LIN {X 0,Y 342.242,Z 667.887,A -85,B 0,C 180,E1 16805.675,E2 16805.675} C_VEL
LIN {X 0,Y 344.093,Z 652.07,A -85,B 0,C 180,E1 16803.884,E2 16803.884} C_VEL
LIN {X 0,Y 345.94,Z 635.37,A -85,B 0,C 180,E1 16802.363,E2 16802.363} C_VEL
LIN {X 0,Y 347.673,Z 617.854,A -85,B 0,C 180,E1 16801.111,E2 16801.111} C_VEL
LIN {X 0,Y 349.271,Z 599.201,A -85,B 0,C 180,E1 16800.115,E2 16800.115} C_VEL
LIN {X 0,Y 350.382,Z 580.027,A -85,B 0,C 180,E1 16799.421,E2 16799.421} C_VEL
LIN {X 0,Y 355.845,Z 417.127,A -85,B 0,C 180,E1 16795.462,E2 16795.462} C_VEL
LIN {X 0,Y 353.483,Z 389.228,A -85,B 0,C 180,E1 16794.516,E2 16794.516} C_VEL
LIN {X 0,Y 357.131,Z 365.009,A -85,B 0,C 180,E1 16791.622,E2 16791.622} C_VEL
LIN {X 0,Y 349.632,Z 342.182,A -85,B 0,C 180,E1 16787.791,E2 16787.791} C_VEL
LIN {X 0,Y 342.112,Z 320.607,A -85,B 0,C 180,E1 16783.792,E2 16783.792} C_VEL
LIN {X 0,Y 337.938,Z 308.703,A -85,B 0,C 180,E1 16781.36,E2 16781.36} C_VEL
LIN {X 0,Y 337.929,Z 308.702,A -85,B 0,C 180,E1 16777.13,E2 16777.13} C_VEL
LIN {X 0,Y 337.924,Z 308.701,A -85,B 0,C 180,E1 16772.83,E2 16772.83} C_VEL
LIN {X 0,Y 337.928,Z 308.701,A -85,B 0,C 180,E1 16768.45,E2 16768.45} C_VEL
LIN {X 0,Y 337.933,Z 308.701,A -85,B 0,C 180,E1 16764.286,E2 16764.286} C_VEL
LIN {X 0,Y 337.943,Z 308.701,A -85,B 0,C 180,E1 16760.074,E2 16760.074} C_VEL
LIN {X 0,Y 337.961,Z 308.701,A -85,B 0,C 180,E1 16755.796,E2 16755.796} C_VEL
LIN {X 0,Y 337.96,Z 308.702,A -85,B 0,C 180,E1 16751.608,E2 16751.608} C_VEL
LIN {X 0,Y 337.954,Z 308.7,A -85,B 0,C 180,E1 16747.311,E2 16747.311} C_VEL
LIN {X 0,Y 337.939,Z 308.699,A -85,B 0,C 180,E1 16743.055,E2 16743.055} C_VEL
LIN {X 0,Y 337.933,Z 308.7,A -85,B 0,C 180,E1 16738.816,E2 16738.816} C_VEL
LIN {X 0,Y 337.931,Z 308.7,A -85,B 0,C 180,E1 16734.57,E2 16734.57} C_VEL
LIN {X 0,Y 337.934,Z 308.699,A -85,B 0,C 180,E1 16730.293,E2 16730.293} C_VEL
LIN {X 0,Y 337.947,Z 308.7,A -85,B 0,C 180,E1 16726.025,E2 16726.025} C_VEL
LIN {X 0,Y 337.963,Z 308.7,A -85,B 0,C 180,E1 16721.727,E2 16721.727} C_VEL
LIN {X 0,Y 337.977,Z 308.698,A -85,B 0,C 180,E1 16717.366,E2 16717.366} C_VEL
LIN {X 0,Y 337.959,Z 308.697,A -85,B 0,C 180,E1 16713.089,E2 16713.089} C_VEL
LIN {X 0,Y 337.958,Z 308.697,A -85,B 0,C 180,E1 16709.021,E2 16709.021} C_VEL
LIN {X 0,Y 337.945,Z 308.698,A -85,B 0,C 180,E1 16704.742,E2 16704.742} C_VEL
LIN {X 0,Y 337.941,Z 308.697,A -85,B 0,C 180,E1 16700.501,E2 16700.501} C_VEL
LIN {X 0,Y 337.944,Z 308.698,A -85,B 0,C 180,E1 16696.19,E2 16696.19} C_VEL
LIN {X 0,Y 337.951,Z 308.699,A -85,B 0,C 180,E1 16691.96,E2 16691.96} C_VEL
LIN {X 0,Y 337.96,Z 308.698,A -85,B 0,C 180,E1 16687.762,E2 16687.762} C_VEL
LIN {X 0,Y 337.98,Z 308.699,A -85,B 0,C 180,E1 16683.382,E2 16683.382} C_VEL
LIN {X 0,Y 337.989,Z 308.696,A -85,B 0,C 180,E1 16679.215,E2 16679.215} C_VEL
LIN {X 0,Y 337.962,Z 308.695,A -85,B 0,C 180,E1 16674.84,E2 16674.84} C_VEL
LIN {X 0,Y 337.954,Z 308.697,A -85,B 0,C 180,E1 16670.612,E2 16670.612} C_VEL
LIN {X 0,Y 337.948,Z 308.697,A -85,B 0,C 180,E1 16666.323,E2 16666.323} C_VEL
LIN {X 0,Y 337.95,Z 308.697,A -85,B 0,C 180,E1 16662.125,E2 16662.125} C_VEL
LIN {X 0,Y 337.957,Z 308.699,A -85,B 0,C 180,E1 16657.82,E2 16657.82} C_VEL
LIN {X 0,Y 337.97,Z 308.699,A -85,B 0,C 180,E1 16653.561,E2 16653.561} C_VEL
LIN {X 0,Y 337.989,Z 308.698,A -85,B 0,C 180,E1 16649.321,E2 16649.321} C_VEL
LIN {X 0,Y 337.976,Z 308.696,A -85,B 0,C 180,E1 16644.907,E2 16644.907} C_VEL
LIN {X 0,Y 337.973,Z 308.695,A -85,B 0,C 180,E1 16640.806,E2 16640.806} C_VEL
LIN {X 0,Y 337.96,Z 308.696,A -85,B 0,C 180,E1 16636.482,E2 16636.482} C_VEL
LIN {X 0,Y 337.959,Z 308.696,A -85,B 0,C 180,E1 16632.257,E2 16632.257} C_VEL
LIN {X 0,Y 337.957,Z 308.698,A -85,B 0,C 180,E1 16627.929,E2 16627.929} C_VEL
LIN {X 0,Y 337.97,Z 308.698,A -85,B 0,C 180,E1 16623.654,E2 16623.654} C_VEL
LIN {X 0,Y 337.982,Z 308.699,A -85,B 0,C 180,E1 16619.407,E2 16619.407} C_VEL
LIN {X 0,Y 337.987,Z 308.698,A -85,B 0,C 180,E1 16615.182,E2 16615.182} C_VEL
LIN {X 0,Y 337.991,Z 308.694,A -85,B 0,C 180,E1 16610.805,E2 16610.805} C_VEL
LIN {X 0,Y 337.978,Z 308.696,A -85,B 0,C 180,E1 16606.658,E2 16606.658} C_VEL
LIN {X 0,Y 337.971,Z 308.699,A -85,B 0,C 180,E1 16602.412,E2 16602.412} C_VEL
LIN {X 0,Y 337.978,Z 308.752,A -85,B 0,C 180,E1 16601.593,E2 16601.593} C_VEL
LIN {X 0,Y 342.926,Z 325.779,A -85,B 0,C 180,E1 16597.751,E2 16597.751} C_VEL
LIN {X 0,Y 347.577,Z 343.263,A -85,B 0,C 180,E1 16594.056,E2 16594.056} C_VEL
LIN {X 0,Y 349.757,Z 352.134,A -85,B 0,C 180,E1 16592.257,E2 16592.257} C_VEL
LIN {X 0,Y 349.677,Z 355.829,A -85,B 0,C 180,E1 16591.603,E2 16591.603} C_VEL
LIN {X 0,Y 347.871,Z 360.579,A -85,B 0,C 180,E1 16590.902,E2 16590.902} C_VEL
LIN {X 0,Y 340.468,Z 373.577,A -85,B 0,C 180,E1 16589.15,E2 16589.15} C_VEL
LIN {X 0,Y 339.309,Z 377.653,A -85,B 0,C 180,E1 16588.506,E2 16588.506} C_VEL
LIN {X 0,Y 336.591,Z 401.793,A -85,B 0,C 180,E1 16584.466,E2 16584.466} C_VEL
LIN {X 0,Y 340.456,Z 436.456,A -85,B 0,C 180,E1 16583.068,E2 16583.068} C_VEL
LIN {X 0,Y 336.471,Z 532.966,A -85,B 0,C 180,E1 16580.059,E2 16580.059} C_VEL
LIN {X 0,Y 335.72,Z 549.826,A -85,B 0,C 180,E1 16579.22,E2 16579.22} C_VEL
LIN {X 0,Y 334.81,Z 566.067,A -85,B 0,C 180,E1 16578.091,E2 16578.091} C_VEL
LIN {X 0,Y 333.738,Z 582.038,A -85,B 0,C 180,E1 16576.622,E2 16576.622} C_VEL
LIN {X 0,Y 332.698,Z 596.678,A -85,B 0,C 180,E1 16574.886,E2 16574.886} C_VEL
LIN {X 0,Y 331.716,Z 609.954,A -85,B 0,C 180,E1 16572.885,E2 16572.885} C_VEL
LIN {X 0,Y 330.934,Z 620.947,A -85,B 0,C 180,E1 16570.794,E2 16570.794} C_VEL
LIN {X 0,Y 330.399,Z 629.807,A -85,B 0,C 180,E1 16568.7,E2 16568.7} C_VEL
LIN {X 0,Y 330.037,Z 637.83,A -85,B 0,C 180,E1 16566.259,E2 16566.259} C_VEL
LIN {X 0,Y 329.915,Z 643.784,A -85,B 0,C 180,E1 16563.82,E2 16563.82} C_VEL
LIN {X 0,Y 330.037,Z 648.132,A -85,B 0,C 180,E1 16561.241,E2 16561.241} C_VEL
LIN {X 0,Y 330.399,Z 650.527,A -85,B 0,C 180,E1 16558.61,E2 16558.61} C_VEL
LIN {X 0,Y 330.992,Z 651.065,A -85,B 0,C 180,E1 16556.187,E2 16556.187} C_VEL
LIN {X 0,Y 331.918,Z 649.726,A -85,B 0,C 180,E1 16553.598,E2 16553.598} C_VEL
LIN {X 0,Y 333.117,Z 646.807,A -85,B 0,C 180,E1 16551.192,E2 16551.192} C_VEL
LIN {X 0,Y 334.647,Z 642.03,A -85,B 0,C 180,E1 16548.799,E2 16548.799} C_VEL
LIN {X 0,Y 336.587,Z 635.419,A -85,B 0,C 180,E1 16546.425,E2 16546.425} C_VEL
LIN {X 0,Y 338.907,Z 626.513,A -85,B 0,C 180,E1 16544.073,E2 16544.073} C_VEL
LIN {X 0,Y 341.25,Z 616.897,A -85,B 0,C 180,E1 16542.08,E2 16542.08} C_VEL
LIN {X 0,Y 343.89,Z 604.887,A -85,B 0,C 180,E1 16540.11,E2 16540.11} C_VEL
LIN {X 0,Y 346.665,Z 591.244,A -85,B 0,C 180,E1 16538.333,E2 16538.333} C_VEL
LIN {X 0,Y 349.446,Z 575.669,A -85,B 0,C 180,E1 16536.741,E2 16536.741} C_VEL
LIN {X 0,Y 351.92,Z 559.982,A -85,B 0,C 180,E1 16535.491,E2 16535.491} C_VEL
LIN {X 0,Y 354.216,Z 542.534,A -85,B 0,C 180,E1 16534.445,E2 16534.445} C_VEL
LIN {X 0,Y 361.198,Z 491.904,A -85,B 0,C 180,E1 16532.223,E2 16532.223} C_VEL
LIN {X 0,Y 367.897,Z 448.392,A -85,B 0,C 180,E1 16530.39,E2 16530.39} C_VEL
LIN {X 0,Y 367.465,Z 432.669,A -85,B 0,C 180,E1 16528.882,E2 16528.882} C_VEL
LIN {X 0,Y 366.778,Z 418.433,A -85,B 0,C 180,E1 16527.238,E2 16527.238} C_VEL
LIN {X 0,Y 366.27,Z 405.199,A -85,B 0,C 180,E1 16525.43,E2 16525.43} C_VEL
LIN {X 0,Y 366.35,Z 400.175,A -85,B 0,C 180,E1 16524.646,E2 16524.646} C_VEL
LIN {X 0,Y 368.778,Z 395.594,A -85,B 0,C 180,E1 16523.573,E2 16523.573} C_VEL
LIN {X 0,Y 369.415,Z 391.695,A -85,B 0,C 180,E1 16521.299,E2 16521.299} C_VEL
LIN {X 0,Y 370.024,Z 389.528,A -85,B 0,C 180,E1 16518.931,E2 16518.931} C_VEL
LIN {X 0,Y 370.832,Z 389.284,A -85,B 0,C 180,E1 16516.495,E2 16516.495} C_VEL
LIN {X 0,Y 371.534,Z 391.679,A -85,B 0,C 180,E1 16513.974,E2 16513.974} C_VEL
LIN {X 0,Y 372.084,Z 395.125,A -85,B 0,C 180,E1 16512.103,E2 16512.103} C_VEL
LIN {X 0,Y 371.235,Z 397.302,A -85,B 0,C 180,E1 16511.78,E2 16511.78} C_VEL
LIN {X 0,Y 371.46,Z 412.671,A -85,B 0,C 180,E1 16510.389,E2 16510.389} C_VEL
LIN {X 0,Y 371.239,Z 424.916,A -85,B 0,C 180,E1 16509.557,E2 16509.557} C_VEL
LIN {X 0,Y 362.025,Z 501.522,A -85,B 0,C 180,E1 16507.037,E2 16507.037} C_VEL
LIN {X 0,Y 354.62,Z 580.346,A -85,B 0,C 180,E1 16504.536,E2 16504.536} C_VEL
LIN {X 0,Y 351.887,Z 599.701,A -85,B 0,C 180,E1 16503.638,E2 16503.638} C_VEL
LIN {X 0,Y 348.616,Z 618.561,A -85,B 0,C 180,E1 16502.436,E2 16502.436} C_VEL
LIN {X 0,Y 345.167,Z 636.473,A -85,B 0,C 180,E1 16500.943,E2 16500.943} C_VEL
LIN {X 0,Y 341.679,Z 653.443,A -85,B 0,C 180,E1 16499.15,E2 16499.15} C_VEL
LIN {X 0,Y 338.323,Z 669.249,A -85,B 0,C 180,E1 16497.074,E2 16497.074} C_VEL
LIN {X 0,Y 335.124,Z 684.622,A -85,B 0,C 180,E1 16494.597,E2 16494.597} C_VEL
LIN {X 0,Y 332.517,Z 698.311,A -85,B 0,C 180,E1 16491.893,E2 16491.893} C_VEL
LIN {X 0,Y 330.578,Z 709.97,A -85,B 0,C 180,E1 16489.067,E2 16489.067} C_VEL
LIN {X 0,Y 329.306,Z 720.112,A -85,B 0,C 180,E1 16486.041,E2 16486.041} C_VEL
LIN {X 0,Y 328.706,Z 728.665,A -85,B 0,C 180,E1 16482.831,E2 16482.831} C_VEL
LIN {X 0,Y 328.709,Z 735.179,A -85,B 0,C 180,E1 16479.632,E2 16479.632} C_VEL
LIN {X 0,Y 329.047,Z 739.533,A -85,B 0,C 180,E1 16476.632,E2 16476.632} C_VEL
LIN {X 0,Y 329.486,Z 742.179,A -85,B 0,C 180,E1 16473.655,E2 16473.655} C_VEL
LIN {X 0,Y 329.775,Z 743.096,A -85,B 0,C 180,E1 16470.87,E2 16470.87} C_VEL
LIN {X 0,Y 329.767,Z 742.439,A -85,B 0,C 180,E1 16468.09,E2 16468.09} C_VEL
LIN {X 0,Y 329.514,Z 740.182,A -85,B 0,C 180,E1 16465.302,E2 16465.302} C_VEL
LIN {X 0,Y 329.182,Z 736.275,A -85,B 0,C 180,E1 16462.497,E2 16462.497} C_VEL
LIN {X 0,Y 328.954,Z 730.625,A -85,B 0,C 180,E1 16459.671,E2 16459.671} C_VEL
LIN {X 0,Y 329.017,Z 723.102,A -85,B 0,C 180,E1 16456.827,E2 16456.827} C_VEL
LIN {X 0,Y 329.447,Z 714.162,A -85,B 0,C 180,E1 16454.15,E2 16454.15} C_VEL
LIN {X 0,Y 330.336,Z 703.098,A -85,B 0,C 180,E1 16451.471,E2 16451.471} C_VEL
LIN {X 0,Y 331.632,Z 690.48,A -85,B 0,C 180,E1 16448.976,E2 16448.976} C_VEL
LIN {X 0,Y 333.279,Z 676.261,A -85,B 0,C 180,E1 16446.673,E2 16446.673} C_VEL
LIN {X 0,Y 335.14,Z 660.941,A -85,B 0,C 180,E1 16444.653,E2 16444.653} C_VEL
LIN {X 0,Y 337.069,Z 644.579,A -85,B 0,C 180,E1 16442.915,E2 16442.915} C_VEL
LIN {X 0,Y 338.953,Z 627.296,A -85,B 0,C 180,E1 16441.455,E2 16441.455} C_VEL
LIN {X 0,Y 340.72,Z 609.034,A -85,B 0,C 180,E1 16440.27,E2 16440.27} C_VEL
LIN {X 0,Y 342.192,Z 590.096,A -85,B 0,C 180,E1 16439.383,E2 16439.383} C_VEL
LIN {X 0,Y 343.081,Z 569.712,A -85,B 0,C 180,E1 16438.771,E2 16438.771} C_VEL
LIN {X 0,Y 348.452,Z 418.182,A -85,B 0,C 180,E1 16434.993,E2 16434.993} C_VEL
LIN {X 0,Y 346.093,Z 389.328,A -85,B 0,C 180,E1 16433.992,E2 16433.992} C_VEL
LIN {X 0,Y 349.501,Z 367.033,A -85,B 0,C 180,E1 16431.259,E2 16431.259} C_VEL
LIN {X 0,Y 342.384,Z 345.277,A -85,B 0,C 180,E1 16427.523,E2 16427.523} C_VEL
LIN {X 0,Y 335.056,Z 324.104,A -85,B 0,C 180,E1 16423.521,E2 16423.521} C_VEL
LIN {X 0,Y 329.981,Z 309.695,A -85,B 0,C 180,E1 16420.539,E2 16420.539} C_VEL
LIN {X 0,Y 329.992,Z 309.692,A -85,B 0,C 180,E1 16416.219,E2 16416.219} C_VEL
LIN {X 0,Y 330.019,Z 309.691,A -85,B 0,C 180,E1 16411.816,E2 16411.816} C_VEL
LIN {X 0,Y 330.02,Z 309.69,A -85,B 0,C 180,E1 16407.618,E2 16407.618} C_VEL
LIN {X 0,Y 330.01,Z 309.69,A -85,B 0,C 180,E1 16403.365,E2 16403.365} C_VEL
LIN {X 0,Y 329.999,Z 309.69,A -85,B 0,C 180,E1 16399.103,E2 16399.103} C_VEL
LIN {X 0,Y 329.986,Z 309.69,A -85,B 0,C 180,E1 16394.747,E2 16394.747} C_VEL
LIN {X 0,Y 329.995,Z 309.69,A -85,B 0,C 180,E1 16390.3,E2 16390.3} C_VEL
LIN {X 0,Y 330.003,Z 309.69,A -85,B 0,C 180,E1 16386.09,E2 16386.09} C_VEL
LIN {X 0,Y 330.022,Z 309.69,A -85,B 0,C 180,E1 16381.739,E2 16381.739} C_VEL
LIN {X 0,Y 330.02,Z 309.688,A -85,B 0,C 180,E1 16377.398,E2 16377.398} C_VEL
LIN {X 0,Y 330.005,Z 309.688,A -85,B 0,C 180,E1 16373.042,E2 16373.042} C_VEL
LIN {X 0,Y 329.998,Z 309.687,A -85,B 0,C 180,E1 16368.822,E2 16368.822} C_VEL
LIN {X 0,Y 329.996,Z 309.689,A -85,B 0,C 180,E1 16364.469,E2 16364.469} C_VEL
LIN {X 0,Y 330.003,Z 309.686,A -85,B 0,C 180,E1 16360.166,E2 16360.166} C_VEL
LIN {X 0,Y 330.008,Z 309.689,A -85,B 0,C 180,E1 16356.05,E2 16356.05} C_VEL
LIN {X 0,Y 330.022,Z 309.687,A -85,B 0,C 180,E1 16351.798,E2 16351.798} C_VEL
LIN {X 0,Y 330.034,Z 309.688,A -85,B 0,C 180,E1 16347.576,E2 16347.576} C_VEL
LIN {X 0,Y 330.025,Z 309.686,A -85,B 0,C 180,E1 16343.144,E2 16343.144} C_VEL
LIN {X 0,Y 330.015,Z 309.683,A -85,B 0,C 180,E1 16338.899,E2 16338.899} C_VEL
LIN {X 0,Y 330.007,Z 309.687,A -85,B 0,C 180,E1 16334.607,E2 16334.607} C_VEL
LIN {X 0,Y 330.006,Z 309.687,A -85,B 0,C 180,E1 16330.19,E2 16330.19} C_VEL
LIN {X 0,Y 330.011,Z 309.684,A -85,B 0,C 180,E1 16325.998,E2 16325.998} C_VEL
LIN {X 0,Y 330.031,Z 309.688,A -85,B 0,C 180,E1 16321.652,E2 16321.652} C_VEL
LIN {X 0,Y 330.044,Z 309.686,A -85,B 0,C 180,E1 16317.416,E2 16317.416} C_VEL
LIN {X 0,Y 330.034,Z 309.684,A -85,B 0,C 180,E1 16313.004,E2 16313.004} C_VEL
LIN {X 0,Y 330.02,Z 309.686,A -85,B 0,C 180,E1 16308.731,E2 16308.731} C_VEL
LIN {X 0,Y 330.009,Z 309.685,A -85,B 0,C 180,E1 16304.384,E2 16304.384} C_VEL
LIN {X 0,Y 330.015,Z 309.687,A -85,B 0,C 180,E1 16299.943,E2 16299.943} C_VEL
LIN {X 0,Y 330.023,Z 309.688,A -85,B 0,C 180,E1 16295.737,E2 16295.737} C_VEL
LIN {X 0,Y 330.041,Z 309.688,A -85,B 0,C 180,E1 16291.387,E2 16291.387} C_VEL
LIN {X 0,Y 330.04,Z 309.684,A -85,B 0,C 180,E1 16287.047,E2 16287.047} C_VEL
LIN {X 0,Y 330.029,Z 309.685,A -85,B 0,C 180,E1 16282.688,E2 16282.688} C_VEL
LIN {X 0,Y 330.019,Z 309.685,A -85,B 0,C 180,E1 16278.464,E2 16278.464} C_VEL
LIN {X 0,Y 330.017,Z 309.685,A -85,B 0,C 180,E1 16274.175,E2 16274.175} C_VEL
LIN {X 0,Y 330.024,Z 309.687,A -85,B 0,C 180,E1 16269.794,E2 16269.794} C_VEL
LIN {X 0,Y 330.029,Z 309.688,A -85,B 0,C 180,E1 16265.666,E2 16265.666} C_VEL
LIN {X 0,Y 330.045,Z 309.688,A -85,B 0,C 180,E1 16261.401,E2 16261.401} C_VEL
LIN {X 0,Y 330.053,Z 309.685,A -85,B 0,C 180,E1 16257.043,E2 16257.043} C_VEL
LIN {X 0,Y 330.042,Z 309.684,A -85,B 0,C 180,E1 16252.705,E2 16252.705} C_VEL
LIN {X 0,Y 330.032,Z 309.685,A -85,B 0,C 180,E1 16248.433,E2 16248.433} C_VEL
LIN {X 0,Y 330.026,Z 309.69,A -85,B 0,C 180,E1 16244.107,E2 16244.107} C_VEL
LIN {X 0,Y 330.047,Z 309.82,A -85,B 0,C 180,E1 16242.293,E2 16242.293} C_VEL
LIN {X 0,Y 335.328,Z 327.903,A -85,B 0,C 180,E1 16238.109,E2 16238.109} C_VEL
LIN {X 0,Y 340.028,Z 345.65,A -85,B 0,C 180,E1 16234.279,E2 16234.279} C_VEL
LIN {X 0,Y 342.178,Z 355.277,A -85,B 0,C 180,E1 16232.322,E2 16232.322} C_VEL
LIN {X 0,Y 339.309,Z 377.653,A -85,B 0,C 180,E1 16228.506,E2 16228.506} C_VEL
LIN {X 0,Y 337.908,Z 381.407,A -85,B 0,C 180,E1 16227.937,E2 16227.937} C_VEL
LIN {X 0,Y 330.822,Z 391.443,A -85,B 0,C 180,E1 16226.626,E2 16226.626} C_VEL
LIN {X 0,Y 329.73,Z 394.679,A -85,B 0,C 180,E1 16226.118,E2 16226.118} C_VEL
LIN {X 0,Y 328.981,Z 401.707,A -85,B 0,C 180,E1 16224.957,E2 16224.957} C_VEL
LIN {X 0,Y 332.841,Z 437.209,A -85,B 0,C 180,E1 16223.481,E2 16223.481} C_VEL
LIN {X 0,Y 328.703,Z 533.627,A -85,B 0,C 180,E1 16220.38,E2 16220.38} C_VEL
LIN {X 0,Y 327.948,Z 550.028,A -85,B 0,C 180,E1 16219.546,E2 16219.546} C_VEL
LIN {X 0,Y 326.976,Z 566.748,A -85,B 0,C 180,E1 16218.356,E2 16218.356} C_VEL
LIN {X 0,Y 325.863,Z 582.787,A -85,B 0,C 180,E1 16216.843,E2 16216.843} C_VEL
LIN {X 0,Y 324.745,Z 598.018,A -85,B 0,C 180,E1 16214.986,E2 16214.986} C_VEL
LIN {X 0,Y 323.745,Z 611.255,A -85,B 0,C 180,E1 16212.936,E2 16212.936} C_VEL
LIN {X 0,Y 322.93,Z 622.663,A -85,B 0,C 180,E1 16210.703,E2 16210.703} C_VEL
LIN {X 0,Y 322.402,Z 631.415,A -85,B 0,C 180,E1 16208.558,E2 16208.558} C_VEL
LIN {X 0,Y 322.064,Z 639.424,A -85,B 0,C 180,E1 16206.056,E2 16206.056} C_VEL
LIN {X 0,Y 321.969,Z 645.288,A -85,B 0,C 180,E1 16203.558,E2 16203.558} C_VEL
LIN {X 0,Y 322.12,Z 649.393,A -85,B 0,C 180,E1 16201.065,E2 16201.065} C_VEL
LIN {X 0,Y 322.531,Z 651.846,A -85,B 0,C 180,E1 16198.399,E2 16198.399} C_VEL
LIN {X 0,Y 323.192,Z 652.469,A -85,B 0,C 180,E1 16195.917,E2 16195.917} C_VEL
LIN {X 0,Y 324.223,Z 651.242,A -85,B 0,C 180,E1 16193.268,E2 16193.268} C_VEL
LIN {X 0,Y 325.534,Z 648.402,A -85,B 0,C 180,E1 16190.807,E2 16190.807} C_VEL
LIN {X 0,Y 327.224,Z 643.805,A -85,B 0,C 180,E1 16188.363,E2 16188.363} C_VEL
LIN {X 0,Y 329.322,Z 637.306,A -85,B 0,C 180,E1 16185.941,E2 16185.941} C_VEL
LIN {X 0,Y 331.657,Z 629.375,A -85,B 0,C 180,E1 16183.716,E2 16183.716} C_VEL
LIN {X 0,Y 334.367,Z 619.283,A -85,B 0,C 180,E1 16181.518,E2 16181.518} C_VEL
LIN {X 0,Y 337.349,Z 607.161,A -85,B 0,C 180,E1 16179.436,E2 16179.436} C_VEL
LIN {X 0,Y 340.615,Z 592.522,A -85,B 0,C 180,E1 16177.474,E2 16177.474} C_VEL
LIN {X 0,Y 343.465,Z 578.024,A -85,B 0,C 180,E1 16175.947,E2 16175.947} C_VEL
LIN {X 0,Y 346.281,Z 561.82,A -85,B 0,C 180,E1 16174.608,E2 16174.608} C_VEL
LIN {X 0,Y 348.857,Z 544.428,A -85,B 0,C 180,E1 16173.52,E2 16173.52} C_VEL
LIN {X 0,Y 355.467,Z 499.569,A -85,B 0,C 180,E1 16171.483,E2 16171.483} C_VEL
LIN {X 0,Y 363.522,Z 450.722,A -85,B 0,C 180,E1 16169.389,E2 16169.389} C_VEL
LIN {X 0,Y 363.468,Z 436.002,A -85,B 0,C 180,E1 16167.918,E2 16167.918} C_VEL
LIN {X 0,Y 363.231,Z 422.494,A -85,B 0,C 180,E1 16166.301,E2 16166.301} C_VEL
LIN {X 0,Y 363.194,Z 409.998,A -85,B 0,C 180,E1 16164.539,E2 16164.539} C_VEL
LIN {X 0,Y 363.472,Z 400.515,A -85,B 0,C 180,E1 16162.954,E2 16162.954} C_VEL
LIN {X 0,Y 363.94,Z 397.554,A -85,B 0,C 180,E1 16161.214,E2 16161.214} C_VEL
LIN {X 0,Y 364.674,Z 395.498,A -85,B 0,C 180,E1 16158.939,E2 16158.939} C_VEL
LIN {X 0,Y 365.497,Z 395.214,A -85,B 0,C 180,E1 16156.633,E2 16156.633} C_VEL
LIN {X 0,Y 366.141,Z 397.534,A -85,B 0,C 180,E1 16154.111,E2 16154.111} C_VEL
LIN {X 0,Y 367.925,Z 401.188,A -85,B 0,C 180,E1 16152.735,E2 16152.735} C_VEL
LIN {X 0,Y 367.706,Z 416.125,A -85,B 0,C 180,E1 16151.346,E2 16151.346} C_VEL
LIN {X 0,Y 367.217,Z 426.833,A -85,B 0,C 180,E1 16150.599,E2 16150.599} C_VEL
LIN {X 0,Y 357.366,Z 500.917,A -85,B 0,C 180,E1 16148.093,E2 16148.093} C_VEL
LIN {X 0,Y 349.11,Z 579.334,A -85,B 0,C 180,E1 16145.506,E2 16145.506} C_VEL
LIN {X 0,Y 346.376,Z 597.432,A -85,B 0,C 180,E1 16144.659,E2 16144.659} C_VEL
LIN {X 0,Y 342.837,Z 616.357,A -85,B 0,C 180,E1 16143.451,E2 16143.451} C_VEL
LIN {X 0,Y 339.114,Z 634.228,A -85,B 0,C 180,E1 16141.956,E2 16141.956} C_VEL
LIN {X 0,Y 335.36,Z 651.175,A -85,B 0,C 180,E1 16140.158,E2 16140.158} C_VEL
LIN {X 0,Y 331.681,Z 667.065,A -85,B 0,C 180,E1 16138.053,E2 16138.053} C_VEL
LIN {X 0,Y 328.265,Z 681.983,A -85,B 0,C 180,E1 16135.629,E2 16135.629} C_VEL
LIN {X 0,Y 325.403,Z 695.384,A -85,B 0,C 180,E1 16132.97,E2 16132.97} C_VEL
LIN {X 0,Y 323.16,Z 707.314,A -85,B 0,C 180,E1 16130.088,E2 16130.088} C_VEL
LIN {X 0,Y 321.607,Z 717.69,A -85,B 0,C 180,E1 16126.993,E2 16126.993} C_VEL
LIN {X 0,Y 320.831,Z 726.031,A -85,B 0,C 180,E1 16123.886,E2 16123.886} C_VEL
LIN {X 0,Y 320.66,Z 732.543,A -85,B 0,C 180,E1 16120.784,E2 16120.784} C_VEL
LIN {X 0,Y 320.939,Z 737.326,A -85,B 0,C 180,E1 16117.7,E2 16117.7} C_VEL
LIN {X 0,Y 321.411,Z 740.407,A -85,B 0,C 180,E1 16114.641,E2 16114.641} C_VEL
LIN {X 0,Y 321.79,Z 741.759,A -85,B 0,C 180,E1 16111.782,E2 16111.782} C_VEL
LIN {X 0,Y 321.918,Z 741.55,A -85,B 0,C 180,E1 16109.112,E2 16109.112} C_VEL
LIN {X 0,Y 321.729,Z 739.777,A -85,B 0,C 180,E1 16106.259,E2 16106.259} C_VEL
LIN {X 0,Y 321.381,Z 736.362,A -85,B 0,C 180,E1 16103.391,E2 16103.391} C_VEL
LIN {X 0,Y 321.083,Z 731.227,A -85,B 0,C 180,E1 16100.502,E2 16100.502} C_VEL
LIN {X 0,Y 321.024,Z 724.256,A -85,B 0,C 180,E1 16097.591,E2 16097.591} C_VEL
LIN {X 0,Y 321.36,Z 715.365,A -85,B 0,C 180,E1 16094.695,E2 16094.695} C_VEL
LIN {X 0,Y 322.159,Z 704.733,A -85,B 0,C 180,E1 16091.92,E2 16091.92} C_VEL
LIN {X 0,Y 323.384,Z 692.644,A -85,B 0,C 180,E1 16089.363,E2 16089.363} C_VEL
LIN {X 0,Y 324.962,Z 679.01,A -85,B 0,C 180,E1 16087,E2 16087} C_VEL
LIN {X 0,Y 326.848,Z 663.752,A -85,B 0,C 180,E1 16084.837,E2 16084.837} C_VEL
LIN {X 0,Y 328.807,Z 647.754,A -85,B 0,C 180,E1 16082.999,E2 16082.999} C_VEL
LIN {X 0,Y 330.729,Z 631.142,A -85,B 0,C 180,E1 16081.469,E2 16081.469} C_VEL
LIN {X 0,Y 332.604,Z 612.794,A -85,B 0,C 180,E1 16080.166,E2 16080.166} C_VEL
LIN {X 0,Y 334.19,Z 594.034,A -85,B 0,C 180,E1 16079.191,E2 16079.191} C_VEL
LIN {X 0,Y 335.235,Z 574.913,A -85,B 0,C 180,E1 16078.52,E2 16078.52} C_VEL
LIN {X 0,Y 340.999,Z 418.598,A -85,B 0,C 180,E1 16074.49,E2 16074.49} C_VEL
LIN {X 0,Y 338.72,Z 389.414,A -85,B 0,C 180,E1 16073.451,E2 16073.451} C_VEL
LIN {X 0,Y 341.939,Z 369.272,A -85,B 0,C 180,E1 16070.929,E2 16070.929} C_VEL
LIN {X 0,Y 335.061,Z 348.183,A -85,B 0,C 180,E1 16067.233,E2 16067.233} C_VEL
LIN {X 0,Y 328.059,Z 327.784,A -85,B 0,C 180,E1 16063.297,E2 16063.297} C_VEL
LIN {X 0,Y 322.082,Z 310.678,A -85,B 0,C 180,E1 16059.659,E2 16059.659} C_VEL
LIN {X 0,Y 322.06,Z 310.68,A -85,B 0,C 180,E1 16055.266,E2 16055.266} C_VEL
LIN {X 0,Y 322.051,Z 310.679,A -85,B 0,C 180,E1 16051.025,E2 16051.025} C_VEL
LIN {X 0,Y 322.048,Z 310.678,A -85,B 0,C 180,E1 16046.604,E2 16046.604} C_VEL
LIN {X 0,Y 322.055,Z 310.68,A -85,B 0,C 180,E1 16042.259,E2 16042.259} C_VEL
LIN {X 0,Y 322.074,Z 310.68,A -85,B 0,C 180,E1 16037.901,E2 16037.901} C_VEL
LIN {X 0,Y 322.089,Z 310.678,A -85,B 0,C 180,E1 16033.649,E2 16033.649} C_VEL
LIN {X 0,Y 322.066,Z 310.676,A -85,B 0,C 180,E1 16029.175,E2 16029.175} C_VEL
LIN {X 0,Y 322.06,Z 310.678,A -85,B 0,C 180,E1 16024.989,E2 16024.989} C_VEL
LIN {X 0,Y 322.052,Z 310.678,A -85,B 0,C 180,E1 16020.536,E2 16020.536} C_VEL
LIN {X 0,Y 322.064,Z 310.676,A -85,B 0,C 180,E1 16016.086,E2 16016.086} C_VEL
LIN {X 0,Y 322.082,Z 310.678,A -85,B 0,C 180,E1 16011.793,E2 16011.793} C_VEL
LIN {X 0,Y 322.09,Z 310.678,A -85,B 0,C 180,E1 16007.452,E2 16007.452} C_VEL
LIN {X 0,Y 322.082,Z 310.675,A -85,B 0,C 180,E1 16003.223,E2 16003.223} C_VEL
LIN {X 0,Y 322.067,Z 310.676,A -85,B 0,C 180,E1 15998.896,E2 15998.896} C_VEL
LIN {X 0,Y 322.061,Z 310.677,A -85,B 0,C 180,E1 15994.608,E2 15994.608} C_VEL
LIN {X 0,Y 322.063,Z 310.672,A -85,B 0,C 180,E1 15990.22,E2 15990.22} C_VEL
LIN {X 0,Y 322.081,Z 310.677,A -85,B 0,C 180,E1 15985.817,E2 15985.817} C_VEL
LIN {X 0,Y 322.108,Z 310.672,A -85,B 0,C 180,E1 15981.401,E2 15981.401} C_VEL
LIN {X 0,Y 322.087,Z 310.674,A -85,B 0,C 180,E1 15977.104,E2 15977.104} C_VEL
LIN {X 0,Y 322.077,Z 310.675,A -85,B 0,C 180,E1 15972.831,E2 15972.831} C_VEL
LIN {X 0,Y 322.068,Z 310.673,A -85,B 0,C 180,E1 15968.531,E2 15968.531} C_VEL
LIN {X 0,Y 322.073,Z 310.674,A -85,B 0,C 180,E1 15964.022,E2 15964.022} C_VEL
LIN {X 0,Y 322.093,Z 310.677,A -85,B 0,C 180,E1 15959.643,E2 15959.643} C_VEL
LIN {X 0,Y 322.1,Z 310.672,A -85,B 0,C 180,E1 15955.363,E2 15955.363} C_VEL
LIN {X 0,Y 322.102,Z 310.674,A -85,B 0,C 180,E1 15951.104,E2 15951.104} C_VEL
LIN {X 0,Y 322.084,Z 310.674,A -85,B 0,C 180,E1 15946.779,E2 15946.779} C_VEL
LIN {X 0,Y 322.076,Z 310.672,A -85,B 0,C 180,E1 15942.55,E2 15942.55} C_VEL
LIN {X 0,Y 322.073,Z 310.677,A -85,B 0,C 180,E1 15938.029,E2 15938.029} C_VEL
LIN {X 0,Y 322.083,Z 310.674,A -85,B 0,C 180,E1 15933.736,E2 15933.736} C_VEL
LIN {X 0,Y 322.112,Z 310.675,A -85,B 0,C 180,E1 15929.287,E2 15929.287} C_VEL
LIN {X 0,Y 322.094,Z 310.673,A -85,B 0,C 180,E1 15924.834,E2 15924.834} C_VEL
LIN {X 0,Y 322.083,Z 310.673,A -85,B 0,C 180,E1 15920.529,E2 15920.529} C_VEL
LIN {X 0,Y 322.077,Z 310.676,A -85,B 0,C 180,E1 15916.169,E2 15916.169} C_VEL
LIN {X 0,Y 322.088,Z 310.676,A -85,B 0,C 180,E1 15911.726,E2 15911.726} C_VEL
LIN {X 0,Y 322.107,Z 310.677,A -85,B 0,C 180,E1 15907.36,E2 15907.36} C_VEL
LIN {X 0,Y 322.111,Z 310.674,A -85,B 0,C 180,E1 15902.975,E2 15902.975} C_VEL
LIN {X 0,Y 322.097,Z 310.673,A -85,B 0,C 180,E1 15898.605,E2 15898.605} C_VEL
LIN {X 0,Y 322.087,Z 310.674,A -85,B 0,C 180,E1 15894.294,E2 15894.294} C_VEL
LIN {X 0,Y 322.086,Z 310.677,A -85,B 0,C 180,E1 15889.78,E2 15889.78} C_VEL
LIN {X 0,Y 322.1,Z 310.679,A -85,B 0,C 180,E1 15885.447,E2 15885.447} C_VEL
LIN {X 0,Y 322.112,Z 310.679,A -85,B 0,C 180,E1 15883.066,E2 15883.066} C_VEL
LIN {X 0,Y 327.284,Z 328.515,A -85,B 0,C 180,E1 15878.827,E2 15878.827} C_VEL
LIN {X 0,Y 332.058,Z 346.254,A -85,B 0,C 180,E1 15874.893,E2 15874.893} C_VEL
LIN {X 0,Y 334.571,Z 357.081,A -85,B 0,C 180,E1 15872.63,E2 15872.63} C_VEL
LIN {X 0,Y 330.98,Z 384.228,A -85,B 0,C 180,E1 15867.917,E2 15867.917} C_VEL
LIN {X 0,Y 329.73,Z 394.679,A -85,B 0,C 180,E1 15866.118,E2 15866.118} C_VEL
LIN {X 0,Y 328.974,Z 399.021,A -85,B 0,C 180,E1 15865.551,E2 15865.551} C_VEL
LIN {X 0,Y 327.242,Z 406.013,A -85,B 0,C 180,E1 15865.046,E2 15865.046} C_VEL
LIN {X 0,Y 324.953,Z 414.646,A -85,B 0,C 180,E1 15864.76,E2 15864.76} C_VEL
LIN {X 0,Y 323.831,Z 421.369,A -85,B 0,C 180,E1 15864.592,E2 15864.592} C_VEL
LIN {X 0,Y 324.229,Z 428.066,A -85,B 0,C 180,E1 15864.327,E2 15864.327} C_VEL
LIN {X 0,Y 325.228,Z 438.303,A -85,B 0,C 180,E1 15863.903,E2 15863.903} C_VEL
LIN {X 0,Y 320.929,Z 533.776,A -85,B 0,C 180,E1 15860.712,E2 15860.712} C_VEL
LIN {X 0,Y 320.104,Z 551.029,A -85,B 0,C 180,E1 15859.807,E2 15859.807} C_VEL
LIN {X 0,Y 319.141,Z 567.163,A -85,B 0,C 180,E1 15858.633,E2 15858.633} C_VEL
LIN {X 0,Y 317.992,Z 583.339,A -85,B 0,C 180,E1 15857.082,E2 15857.082} C_VEL
LIN {X 0,Y 316.841,Z 598.677,A -85,B 0,C 180,E1 15855.181,E2 15855.181} C_VEL
LIN {X 0,Y 315.773,Z 612.545,A -85,B 0,C 180,E1 15852.989,E2 15852.989} C_VEL
LIN {X 0,Y 314.925,Z 624.39,A -85,B 0,C 180,E1 15850.608,E2 15850.608} C_VEL
LIN {X 0,Y 314.373,Z 633.64,A -85,B 0,C 180,E1 15848.226,E2 15848.226} C_VEL
LIN {X 0,Y 314.085,Z 640.926,A -85,B 0,C 180,E1 15845.844,E2 15845.844} C_VEL
LIN {X 0,Y 314.034,Z 647.136,A -85,B 0,C 180,E1 15843.1,E2 15843.1} C_VEL
LIN {X 0,Y 314.245,Z 651.042,A -85,B 0,C 180,E1 15840.544,E2 15840.544} C_VEL
LIN {X 0,Y 314.756,Z 653.389,A -85,B 0,C 180,E1 15837.813,E2 15837.813} C_VEL
LIN {X 0,Y 315.528,Z 653.832,A -85,B 0,C 180,E1 15835.272,E2 15835.272} C_VEL
LIN {X 0,Y 316.725,Z 652.498,A -85,B 0,C 180,E1 15832.561,E2 15832.561} C_VEL
LIN {X 0,Y 318.224,Z 649.552,A -85,B 0,C 180,E1 15830.046,E2 15830.046} C_VEL
LIN {X 0,Y 320.282,Z 644.421,A -85,B 0,C 180,E1 15827.375,E2 15827.375} C_VEL
LIN {X 0,Y 322.482,Z 638.267,A -85,B 0,C 180,E1 15825.085,E2 15825.085} C_VEL
LIN {X 0,Y 325.502,Z 628.849,A -85,B 0,C 180,E1 15822.478,E2 15822.478} C_VEL
LIN {X 0,Y 328.539,Z 618.325,A -85,B 0,C 180,E1 15820.254,E2 15820.254} C_VEL
LIN {X 0,Y 331.733,Z 606.328,A -85,B 0,C 180,E1 15818.237,E2 15818.237} C_VEL
LIN {X 0,Y 335.022,Z 592.681,A -85,B 0,C 180,E1 15816.425,E2 15816.425} C_VEL
LIN {X 0,Y 338.494,Z 576.538,A -85,B 0,C 180,E1 15814.731,E2 15814.731} C_VEL
LIN {X 0,Y 341.597,Z 559.959,A -85,B 0,C 180,E1 15813.393,E2 15813.393} C_VEL
LIN {X 0,Y 344.538,Z 541.125,A -85,B 0,C 180,E1 15812.266,E2 15812.266} C_VEL
LIN {X 0,Y 359.462,Z 453.035,A -85,B 0,C 180,E1 15808.339,E2 15808.339} C_VEL
LIN {X 0,Y 359.776,Z 438.869,A -85,B 0,C 180,E1 15806.863,E2 15806.863} C_VEL
LIN {X 0,Y 360.042,Z 424.829,A -85,B 0,C 180,E1 15805.103,E2 15805.103} C_VEL
LIN {X 0,Y 360.661,Z 410.978,A -85,B 0,C 180,E1 15803.014,E2 15803.014} C_VEL
LIN {X 0,Y 360.921,Z 407.068,A -85,B 0,C 180,E1 15802.302,E2 15802.302} C_VEL
LIN {X 0,Y 360.471,Z 403.505,A -85,B 0,C 180,E1 15800.151,E2 15800.151} C_VEL
LIN {X 0,Y 360.704,Z 402.269,A -85,B 0,C 180,E1 15798.507,E2 15798.507} C_VEL
LIN {X 0,Y 361.695,Z 402.266,A -85,B 0,C 180,E1 15796.639,E2 15796.639} C_VEL
LIN {X 0,Y 363.773,Z 404.998,A -85,B 0,C 180,E1 15794.385,E2 15794.385} C_VEL
LIN {X 0,Y 364.799,Z 407.334,A -85,B 0,C 180,E1 15793.487,E2 15793.487} C_VEL
LIN {X 0,Y 364.101,Z 421.647,A -85,B 0,C 180,E1 15792.168,E2 15792.168} C_VEL
LIN {X 0,Y 363.511,Z 429.077,A -85,B 0,C 180,E1 15791.673,E2 15791.673} C_VEL
LIN {X 0,Y 352.858,Z 501.719,A -85,B 0,C 180,E1 15789.152,E2 15789.152} C_VEL
LIN {X 0,Y 343.797,Z 579.015,A -85,B 0,C 180,E1 15786.509,E2 15786.509} C_VEL
LIN {X 0,Y 340.509,Z 598.458,A -85,B 0,C 180,E1 15785.55,E2 15785.55} C_VEL
LIN {X 0,Y 336.57,Z 617.693,A -85,B 0,C 180,E1 15784.262,E2 15784.262} C_VEL
LIN {X 0,Y 332.651,Z 634.899,A -85,B 0,C 180,E1 15782.755,E2 15782.755} C_VEL
LIN {X 0,Y 328.53,Z 651.755,A -85,B 0,C 180,E1 15780.877,E2 15780.877} C_VEL
LIN {X 0,Y 324.456,Z 667.932,A -85,B 0,C 180,E1 15778.634,E2 15778.634} C_VEL
LIN {X 0,Y 320.853,Z 682.406,A -85,B 0,C 180,E1 15776.168,E2 15776.168} C_VEL
LIN {X 0,Y 317.895,Z 695.062,A -85,B 0,C 180,E1 15773.545,E2 15773.545} C_VEL
LIN {X 0,Y 315.466,Z 706.721,A -85,B 0,C 180,E1 15770.599,E2 15770.599} C_VEL
LIN {X 0,Y 313.758,Z 716.897,A -85,B 0,C 180,E1 15767.432,E2 15767.432} C_VEL
LIN {X 0,Y 312.856,Z 725.528,A -85,B 0,C 180,E1 15764.058,E2 15764.058} C_VEL
LIN {X 0,Y 312.68,Z 732.152,A -85,B 0,C 180,E1 15760.69,E2 15760.69} C_VEL
LIN {X 0,Y 313.005,Z 736.638,A -85,B 0,C 180,E1 15757.527,E2 15757.527} C_VEL
LIN {X 0,Y 313.53,Z 739.433,A -85,B 0,C 180,E1 15754.391,E2 15754.391} C_VEL
LIN {X 0,Y 313.93,Z 740.487,A -85,B 0,C 180,E1 15751.461,E2 15751.461} C_VEL
LIN {X 0,Y 314.018,Z 740.048,A -85,B 0,C 180,E1 15748.724,E2 15748.724} C_VEL
LIN {X 0,Y 313.793,Z 737.987,A -85,B 0,C 180,E1 15745.799,E2 15745.799} C_VEL
LIN {X 0,Y 313.404,Z 734.219,A -85,B 0,C 180,E1 15742.845,E2 15742.845} C_VEL
LIN {X 0,Y 313.113,Z 728.711,A -85,B 0,C 180,E1 15739.886,E2 15739.886} C_VEL
LIN {X 0,Y 313.123,Z 721.27,A -85,B 0,C 180,E1 15736.892,E2 15736.892} C_VEL
LIN {X 0,Y 313.531,Z 712.423,A -85,B 0,C 180,E1 15734.084,E2 15734.084} C_VEL
LIN {X 0,Y 314.433,Z 701.415,A -85,B 0,C 180,E1 15731.268,E2 15731.268} C_VEL
LIN {X 0,Y 315.776,Z 688.836,A -85,B 0,C 180,E1 15728.648,E2 15728.648} C_VEL
LIN {X 0,Y 317.425,Z 675.232,A -85,B 0,C 180,E1 15726.323,E2 15726.323} C_VEL
LIN {X 0,Y 319.359,Z 660.11,A -85,B 0,C 180,E1 15724.205,E2 15724.205} C_VEL
LIN {X 0,Y 321.371,Z 643.951,A -85,B 0,C 180,E1 15722.384,E2 15722.384} C_VEL
LIN {X 0,Y 323.336,Z 626.922,A -85,B 0,C 180,E1 15720.855,E2 15720.855} C_VEL
LIN {X 0,Y 325.244,Z 608.329,A -85,B 0,C 180,E1 15719.573,E2 15719.573} C_VEL
LIN {X 0,Y 326.801,Z 589.547,A -85,B 0,C 180,E1 15718.633,E2 15718.633} C_VEL
LIN {X 0,Y 327.757,Z 569.637,A -85,B 0,C 180,E1 15717.984,E2 15717.984} C_VEL
LIN {X 0,Y 333.578,Z 419.401,A -85,B 0,C 180,E1 15713.992,E2 15713.992} C_VEL
LIN {X 0,Y 331.364,Z 389.357,A -85,B 0,C 180,E1 15712.882,E2 15712.882} C_VEL
LIN {X 0,Y 334.36,Z 371.432,A -85,B 0,C 180,E1 15710.58,E2 15710.58} C_VEL
LIN {X 0,Y 327.409,Z 350.12,A -85,B 0,C 180,E1 15706.75,E2 15706.75} C_VEL
LIN {X 0,Y 320.332,Z 329.314,A -85,B 0,C 180,E1 15702.637,E2 15702.637} C_VEL
LIN {X 0,Y 314.106,Z 311.673,A -85,B 0,C 180,E1 15698.753,E2 15698.753} C_VEL
LIN {X 0,Y 314.114,Z 311.67,A -85,B 0,C 180,E1 15694.294,E2 15694.294} C_VEL
LIN {X 0,Y 314.147,Z 311.668,A -85,B 0,C 180,E1 15689.772,E2 15689.772} C_VEL
LIN {X 0,Y 314.129,Z 311.669,A -85,B 0,C 180,E1 15685.32,E2 15685.32} C_VEL
LIN {X 0,Y 314.113,Z 311.667,A -85,B 0,C 180,E1 15680.888,E2 15680.888} C_VEL
LIN {X 0,Y 314.112,Z 311.667,A -85,B 0,C 180,E1 15676.459,E2 15676.459} C_VEL
LIN {X 0,Y 314.122,Z 311.667,A -85,B 0,C 180,E1 15672.129,E2 15672.129} C_VEL
LIN {X 0,Y 314.152,Z 311.666,A -85,B 0,C 180,E1 15667.684,E2 15667.684} C_VEL
LIN {X 0,Y 314.133,Z 311.666,A -85,B 0,C 180,E1 15663.287,E2 15663.287} C_VEL
LIN {X 0,Y 314.122,Z 311.666,A -85,B 0,C 180,E1 15658.908,E2 15658.908} C_VEL
LIN {X 0,Y 314.117,Z 311.667,A -85,B 0,C 180,E1 15654.34,E2 15654.34} C_VEL
LIN {X 0,Y 314.134,Z 311.665,A -85,B 0,C 180,E1 15649.921,E2 15649.921} C_VEL
LIN {X 0,Y 314.16,Z 311.666,A -85,B 0,C 180,E1 15645.441,E2 15645.441} C_VEL
LIN {X 0,Y 314.131,Z 311.661,A -85,B 0,C 180,E1 15640.962,E2 15640.962} C_VEL
LIN {X 0,Y 314.122,Z 311.666,A -85,B 0,C 180,E1 15636.558,E2 15636.558} C_VEL
LIN {X 0,Y 314.131,Z 311.664,A -85,B 0,C 180,E1 15632.106,E2 15632.106} C_VEL
LIN {X 0,Y 314.15,Z 311.664,A -85,B 0,C 180,E1 15627.68,E2 15627.68} C_VEL
LIN {X 0,Y 314.15,Z 311.664,A -85,B 0,C 180,E1 15623.252,E2 15623.252} C_VEL
LIN {X 0,Y 314.14,Z 311.658,A -85,B 0,C 180,E1 15618.965,E2 15618.965} C_VEL
LIN {X 0,Y 314.129,Z 311.664,A -85,B 0,C 180,E1 15614.445,E2 15614.445} C_VEL
LIN {X 0,Y 314.133,Z 311.665,A -85,B 0,C 180,E1 15610.01,E2 15610.01} C_VEL
LIN {X 0,Y 314.149,Z 311.66,A -85,B 0,C 180,E1 15605.621,E2 15605.621} C_VEL
LIN {X 0,Y 314.159,Z 311.664,A -85,B 0,C 180,E1 15601.122,E2 15601.122} C_VEL
LIN {X 0,Y 314.146,Z 311.661,A -85,B 0,C 180,E1 15596.867,E2 15596.867} C_VEL
LIN {X 0,Y 314.135,Z 311.661,A -85,B 0,C 180,E1 15592.453,E2 15592.453} C_VEL
LIN {X 0,Y 314.14,Z 311.666,A -85,B 0,C 180,E1 15587.898,E2 15587.898} C_VEL
LIN {X 0,Y 314.151,Z 311.662,A -85,B 0,C 180,E1 15583.621,E2 15583.621} C_VEL
LIN {X 0,Y 314.164,Z 311.664,A -85,B 0,C 180,E1 15579.155,E2 15579.155} C_VEL
LIN {X 0,Y 314.144,Z 311.66,A -85,B 0,C 180,E1 15574.745,E2 15574.745} C_VEL
LIN {X 0,Y 314.138,Z 311.664,A -85,B 0,C 180,E1 15570.363,E2 15570.363} C_VEL
LIN {X 0,Y 314.142,Z 311.663,A -85,B 0,C 180,E1 15565.801,E2 15565.801} C_VEL
LIN {X 0,Y 314.164,Z 311.666,A -85,B 0,C 180,E1 15561.396,E2 15561.396} C_VEL
LIN {X 0,Y 314.162,Z 311.663,A -85,B 0,C 180,E1 15556.859,E2 15556.859} C_VEL
LIN {X 0,Y 314.151,Z 311.662,A -85,B 0,C 180,E1 15552.59,E2 15552.59} C_VEL
LIN {X 0,Y 314.141,Z 311.664,A -85,B 0,C 180,E1 15548.135,E2 15548.135} C_VEL
LIN {X 0,Y 314.151,Z 311.665,A -85,B 0,C 180,E1 15543.741,E2 15543.741} C_VEL
LIN {X 0,Y 314.167,Z 311.667,A -85,B 0,C 180,E1 15539.387,E2 15539.387} C_VEL
LIN {X 0,Y 314.169,Z 311.664,A -85,B 0,C 180,E1 15535.049,E2 15535.049} C_VEL
LIN {X 0,Y 314.163,Z 311.663,A -85,B 0,C 180,E1 15530.652,E2 15530.652} C_VEL
LIN {X 0,Y 314.151,Z 311.666,A -85,B 0,C 180,E1 15526.255,E2 15526.255} C_VEL
LIN {X 0,Y 314.178,Z 311.864,A -85,B 0,C 180,E1 15523.795,E2 15523.795} C_VEL
LIN {X 0,Y 319.082,Z 328.444,A -85,B 0,C 180,E1 15519.731,E2 15519.731} C_VEL
LIN {X 0,Y 323.698,Z 345.555,A -85,B 0,C 180,E1 15515.821,E2 15515.821} C_VEL
LIN {X 0,Y 326.9,Z 359.243,A -85,B 0,C 180,E1 15512.878,E2 15512.878} C_VEL
LIN {X 0,Y 323.155,Z 386.556,A -85,B 0,C 180,E1 15508.05,E2 15508.05} C_VEL
LIN {X 0,Y 321.378,Z 401.64,A -85,B 0,C 180,E1 15505.456,E2 15505.456} C_VEL
LIN {X 0,Y 324.229,Z 428.066,A -85,B 0,C 180,E1 15504.327,E2 15504.327} C_VEL
LIN {X 0,Y 323.89,Z 432.416,A -85,B 0,C 180,E1 15504.192,E2 15504.192} C_VEL
LIN {X 0,Y 321.097,Z 439.406,A -85,B 0,C 180,E1 15504.105,E2 15504.105} C_VEL
LIN {X 0,Y 317.672,Z 447.141,A -85,B 0,C 180,E1 15504.027,E2 15504.027} C_VEL
LIN {X 0,Y 316.993,Z 450.842,A -85,B 0,C 180,E1 15503.932,E2 15503.932} C_VEL
LIN {X 0,Y 313.124,Z 534.817,A -85,B 0,C 180,E1 15501.016,E2 15501.016} C_VEL
LIN {X 0,Y 312.302,Z 551.436,A -85,B 0,C 180,E1 15500.12,E2 15500.12} C_VEL
LIN {X 0,Y 311.313,Z 567.571,A -85,B 0,C 180,E1 15498.925,E2 15498.925} C_VEL
LIN {X 0,Y 310.135,Z 583.755,A -85,B 0,C 180,E1 15497.347,E2 15497.347} C_VEL
LIN {X 0,Y 308.99,Z 598.612,A -85,B 0,C 180,E1 15495.48,E2 15495.48} C_VEL
LIN {X 0,Y 307.957,Z 611.61,A -85,B 0,C 180,E1 15493.42,E2 15493.42} C_VEL
LIN {X 0,Y 307.134,Z 622.615,A -85,B 0,C 180,E1 15491.261,E2 15491.261} C_VEL
LIN {X 0,Y 306.509,Z 632.59,A -85,B 0,C 180,E1 15488.816,E2 15488.816} C_VEL
LIN {X 0,Y 306.145,Z 640.901,A -85,B 0,C 180,E1 15486.184,E2 15486.184} C_VEL
LIN {X 0,Y 306.066,Z 646.797,A -85,B 0,C 180,E1 15483.743,E2 15483.743} C_VEL
LIN {X 0,Y 306.256,Z 651.538,A -85,B 0,C 180,E1 15480.933,E2 15480.933} C_VEL
LIN {X 0,Y 306.718,Z 654.248,A -85,B 0,C 180,E1 15478.316,E2 15478.316} C_VEL
LIN {X 0,Y 307.548,Z 655.284,A -85,B 0,C 180,E1 15475.522,E2 15475.522} C_VEL
LIN {X 0,Y 308.695,Z 654.609,A -85,B 0,C 180,E1 15472.928,E2 15472.928} C_VEL
LIN {X 0,Y 310.327,Z 651.985,A -85,B 0,C 180,E1 15470.165,E2 15470.165} C_VEL
LIN {X 0,Y 312.325,Z 647.877,A -85,B 0,C 180,E1 15467.612,E2 15467.612} C_VEL
LIN {X 0,Y 314.754,Z 641.864,A -85,B 0,C 180,E1 15465.087,E2 15465.087} C_VEL
LIN {X 0,Y 317.688,Z 633.954,A -85,B 0,C 180,E1 15462.601,E2 15462.601} C_VEL
LIN {X 0,Y 321.36,Z 622.865,A -85,B 0,C 180,E1 15459.984,E2 15459.984} C_VEL
LIN {X 0,Y 324.984,Z 610.598,A -85,B 0,C 180,E1 15457.762,E2 15457.762} C_VEL
LIN {X 0,Y 328.632,Z 597.199,A -85,B 0,C 180,E1 15455.842,E2 15455.842} C_VEL
LIN {X 0,Y 332.306,Z 582.125,A -85,B 0,C 180,E1 15454.131,E2 15454.131} C_VEL
LIN {X 0,Y 335.764,Z 566.013,A -85,B 0,C 180,E1 15452.702,E2 15452.702} C_VEL
LIN {X 0,Y 339.013,Z 548.186,A -85,B 0,C 180,E1 15451.505,E2 15451.505} C_VEL
LIN {X 0,Y 345.398,Z 510.553,A -85,B 0,C 180,E1 15449.693,E2 15449.693} C_VEL
LIN {X 0,Y 355.74,Z 455.471,A -85,B 0,C 180,E1 15447.255,E2 15447.255} C_VEL
LIN {X 0,Y 356.437,Z 441.635,A -85,B 0,C 180,E1 15445.75,E2 15445.75} C_VEL
LIN {X 0,Y 357.219,Z 427.962,A -85,B 0,C 180,E1 15443.948,E2 15443.948} C_VEL
LIN {X 0,Y 358.323,Z 415.673,A -85,B 0,C 180,E1 15442.026,E2 15442.026} C_VEL
LIN {X 0,Y 358.505,Z 413.696,A -85,B 0,C 180,E1 15441.602,E2 15441.602} C_VEL
LIN {X 0,Y 358.409,Z 410.791,A -85,B 0,C 180,E1 15439.606,E2 15439.606} C_VEL
LIN {X 0,Y 358.864,Z 409.906,A -85,B 0,C 180,E1 15438.033,E2 15438.033} C_VEL
LIN {X 0,Y 359.771,Z 410.183,A -85,B 0,C 180,E1 15436.5,E2 15436.5} C_VEL
LIN {X 0,Y 361.493,Z 412.619,A -85,B 0,C 180,E1 15434.593,E2 15434.593} C_VEL
LIN {X 0,Y 361.806,Z 413.681,A -85,B 0,C 180,E1 15434.24,E2 15434.24} C_VEL
LIN {X 0,Y 360.734,Z 426.993,A -85,B 0,C 180,E1 15433.044,E2 15433.044} C_VEL
LIN {X 0,Y 360.192,Z 431.376,A -85,B 0,C 180,E1 15432.785,E2 15432.785} C_VEL
LIN {X 0,Y 348.665,Z 502.796,A -85,B 0,C 180,E1 15430.251,E2 15430.251} C_VEL
LIN {X 0,Y 338.876,Z 577.9,A -85,B 0,C 180,E1 15427.599,E2 15427.599} C_VEL
LIN {X 0,Y 335.541,Z 596.23,A -85,B 0,C 180,E1 15426.689,E2 15426.689} C_VEL
LIN {X 0,Y 331.314,Z 615.339,A -85,B 0,C 180,E1 15425.412,E2 15425.412} C_VEL
LIN {X 0,Y 327.016,Z 632.852,A -85,B 0,C 180,E1 15423.874,E2 15423.874} C_VEL
LIN {X 0,Y 322.592,Z 649.549,A -85,B 0,C 180,E1 15422.007,E2 15422.007} C_VEL
LIN {X 0,Y 318.197,Z 665.579,A -85,B 0,C 180,E1 15419.769,E2 15419.769} C_VEL
LIN {X 0,Y 314.222,Z 680.1,A -85,B 0,C 180,E1 15417.273,E2 15417.273} C_VEL
LIN {X 0,Y 310.66,Z 693.834,A -85,B 0,C 180,E1 15414.375,E2 15414.375} C_VEL
LIN {X 0,Y 307.867,Z 705.847,A -85,B 0,C 180,E1 15411.233,E2 15411.233} C_VEL
LIN {X 0,Y 305.929,Z 716.164,A -85,B 0,C 180,E1 15407.893,E2 15407.893} C_VEL
LIN {X 0,Y 304.914,Z 724.646,A -85,B 0,C 180,E1 15404.432,E2 15404.432} C_VEL
LIN {X 0,Y 304.686,Z 731.146,A -85,B 0,C 180,E1 15400.974,E2 15400.974} C_VEL
LIN {X 0,Y 305.014,Z 735.525,A -85,B 0,C 180,E1 15397.725,E2 15397.725} C_VEL
LIN {X 0,Y 305.577,Z 738.225,A -85,B 0,C 180,E1 15394.505,E2 15394.505} C_VEL
LIN {X 0,Y 306.031,Z 739.181,A -85,B 0,C 180,E1 15391.499,E2 15391.499} C_VEL
LIN {X 0,Y 306.139,Z 738.631,A -85,B 0,C 180,E1 15388.691,E2 15388.691} C_VEL
LIN {X 0,Y 305.919,Z 736.64,A -85,B 0,C 180,E1 15385.878,E2 15385.878} C_VEL
LIN {X 0,Y 305.508,Z 732.84,A -85,B 0,C 180,E1 15382.857,E2 15382.857} C_VEL
LIN {X 0,Y 305.195,Z 727.25,A -85,B 0,C 180,E1 15379.812,E2 15379.812} C_VEL
LIN {X 0,Y 305.204,Z 719.742,A -85,B 0,C 180,E1 15376.744,E2 15376.744} C_VEL
LIN {X 0,Y 305.626,Z 710.773,A -85,B 0,C 180,E1 15373.856,E2 15373.856} C_VEL
LIN {X 0,Y 306.574,Z 699.642,A -85,B 0,C 180,E1 15370.967,E2 15370.967} C_VEL
LIN {X 0,Y 307.918,Z 687.415,A -85,B 0,C 180,E1 15368.378,E2 15368.378} C_VEL
LIN {X 0,Y 309.624,Z 673.698,A -85,B 0,C 180,E1 15365.992,E2 15365.992} C_VEL
LIN {X 0,Y 311.623,Z 658.393,A -85,B 0,C 180,E1 15363.823,E2 15363.823} C_VEL
LIN {X 0,Y 313.694,Z 642.132,A -85,B 0,C 180,E1 15361.969,E2 15361.969} C_VEL
LIN {X 0,Y 315.739,Z 624.779,A -85,B 0,C 180,E1 15360.397,E2 15360.397} C_VEL
LIN {X 0,Y 317.63,Z 606.573,A -85,B 0,C 180,E1 15359.131,E2 15359.131} C_VEL
LIN {X 0,Y 319.2,Z 587.774,A -85,B 0,C 180,E1 15358.188,E2 15358.188} C_VEL
LIN {X 0,Y 320.198,Z 566.554,A -85,B 0,C 180,E1 15357.499,E2 15357.499} C_VEL
LIN {X 0,Y 326.142,Z 420.086,A -85,B 0,C 180,E1 15353.482,E2 15353.482} C_VEL
LIN {X 0,Y 323.973,Z 389.573,A -85,B 0,C 180,E1 15352.335,E2 15352.335} C_VEL
LIN {X 0,Y 326.694,Z 373.335,A -85,B 0,C 180,E1 15350.194,E2 15350.194} C_VEL
LIN {X 0,Y 319.416,Z 350.951,A -85,B 0,C 180,E1 15346.054,E2 15346.054} C_VEL
LIN {X 0,Y 312.871,Z 331.792,A -85,B 0,C 180,E1 15342.15,E2 15342.15} C_VEL
LIN {X 0,Y 306.978,Z 315.299,A -85,B 0,C 180,E1 15338.472,E2 15338.472} C_VEL
LIN {X 0,Y 306.196,Z 312.657,A -85,B 0,C 180,E1 15337.874,E2 15337.874} C_VEL
LIN {X 0,Y 306.197,Z 312.657,A -85,B 0,C 180,E1 15333.497,E2 15333.497} C_VEL
LIN {X 0,Y 306.174,Z 312.657,A -85,B 0,C 180,E1 15328.935,E2 15328.935} C_VEL
LIN {X 0,Y 306.178,Z 312.658,A -85,B 0,C 180,E1 15324.299,E2 15324.299} C_VEL
LIN {X 0,Y 306.198,Z 312.657,A -85,B 0,C 180,E1 15319.855,E2 15319.855} C_VEL
LIN {X 0,Y 306.196,Z 312.656,A -85,B 0,C 180,E1 15315.34,E2 15315.34} C_VEL
LIN {X 0,Y 306.177,Z 312.657,A -85,B 0,C 180,E1 15310.921,E2 15310.921} C_VEL
LIN {X 0,Y 306.176,Z 312.657,A -85,B 0,C 180,E1 15306.377,E2 15306.377} C_VEL
LIN {X 0,Y 306.197,Z 312.655,A -85,B 0,C 180,E1 15301.874,E2 15301.874} C_VEL
LIN {X 0,Y 306.204,Z 312.653,A -85,B 0,C 180,E1 15297.57,E2 15297.57} C_VEL
LIN {X 0,Y 306.19,Z 312.655,A -85,B 0,C 180,E1 15293.061,E2 15293.061} C_VEL
LIN {X 0,Y 306.178,Z 312.653,A -85,B 0,C 180,E1 15288.513,E2 15288.513} C_VEL
LIN {X 0,Y 306.189,Z 312.656,A -85,B 0,C 180,E1 15284.083,E2 15284.083} C_VEL
LIN {X 0,Y 306.214,Z 312.652,A -85,B 0,C 180,E1 15279.554,E2 15279.554} C_VEL
LIN {X 0,Y 306.201,Z 312.654,A -85,B 0,C 180,E1 15275.091,E2 15275.091} C_VEL
LIN {X 0,Y 306.186,Z 312.647,A -85,B 0,C 180,E1 15270.675,E2 15270.675} C_VEL
LIN {X 0,Y 306.193,Z 312.654,A -85,B 0,C 180,E1 15266.059,E2 15266.059} C_VEL
LIN {X 0,Y 306.217,Z 312.652,A -85,B 0,C 180,E1 15261.593,E2 15261.593} C_VEL
LIN {X 0,Y 306.213,Z 312.651,A -85,B 0,C 180,E1 15257.226,E2 15257.226} C_VEL
LIN {X 0,Y 306.195,Z 312.653,A -85,B 0,C 180,E1 15252.722,E2 15252.722} C_VEL
LIN {X 0,Y 306.192,Z 312.65,A -85,B 0,C 180,E1 15248.102,E2 15248.102} C_VEL
LIN {X 0,Y 306.212,Z 312.652,A -85,B 0,C 180,E1 15243.636,E2 15243.636} C_VEL
LIN {X 0,Y 306.222,Z 312.651,A -85,B 0,C 180,E1 15239.109,E2 15239.109} C_VEL
LIN {X 0,Y 306.201,Z 312.645,A -85,B 0,C 180,E1 15234.705,E2 15234.705} C_VEL
LIN {X 0,Y 306.195,Z 312.653,A -85,B 0,C 180,E1 15230.249,E2 15230.249} C_VEL
LIN {X 0,Y 306.208,Z 312.653,A -85,B 0,C 180,E1 15225.723,E2 15225.723} C_VEL
LIN {X 0,Y 306.222,Z 312.654,A -85,B 0,C 180,E1 15221.296,E2 15221.296} C_VEL
LIN {X 0,Y 306.208,Z 312.651,A -85,B 0,C 180,E1 15216.749,E2 15216.749} C_VEL
LIN {X 0,Y 306.197,Z 312.651,A -85,B 0,C 180,E1 15212.244,E2 15212.244} C_VEL
LIN {X 0,Y 306.206,Z 312.654,A -85,B 0,C 180,E1 15207.753,E2 15207.753} C_VEL
LIN {X 0,Y 306.235,Z 312.653,A -85,B 0,C 180,E1 15203.248,E2 15203.248} C_VEL
LIN {X 0,Y 306.212,Z 312.651,A -85,B 0,C 180,E1 15198.7,E2 15198.7} C_VEL
LIN {X 0,Y 306.203,Z 312.651,A -85,B 0,C 180,E1 15194.273,E2 15194.273} C_VEL
LIN {X 0,Y 306.21,Z 312.654,A -85,B 0,C 180,E1 15189.748,E2 15189.748} C_VEL
LIN {X 0,Y 306.226,Z 312.653,A -85,B 0,C 180,E1 15185.294,E2 15185.294} C_VEL
LIN {X 0,Y 306.235,Z 312.651,A -85,B 0,C 180,E1 15180.889,E2 15180.889} C_VEL
LIN {X 0,Y 306.21,Z 312.652,A -85,B 0,C 180,E1 15176.365,E2 15176.365} C_VEL
LIN {X 0,Y 306.209,Z 312.655,A -85,B 0,C 180,E1 15171.891,E2 15171.891} C_VEL
LIN {X 0,Y 306.221,Z 312.657,A -85,B 0,C 180,E1 15167.475,E2 15167.475} C_VEL
LIN {X 0,Y 306.237,Z 312.758,A -85,B 0,C 180,E1 15164.619,E2 15164.619} C_VEL
LIN {X 0,Y 311.321,Z 329.99,A -85,B 0,C 180,E1 15160.275,E2 15160.275} C_VEL
LIN {X 0,Y 315.738,Z 346.291,A -85,B 0,C 180,E1 15156.45,E2 15156.45} C_VEL
LIN {X 0,Y 319.307,Z 360.911,A -85,B 0,C 180,E1 15153.225,E2 15153.225} C_VEL
LIN {X 0,Y 315.392,Z 388.299,A -85,B 0,C 180,E1 15148.287,E2 15148.287} C_VEL
LIN {X 0,Y 313.779,Z 401.534,A -85,B 0,C 180,E1 15145.971,E2 15145.971} C_VEL
LIN {X 0,Y 317.598,Z 438.97,A -85,B 0,C 180,E1 15144.328,E2 15144.328} C_VEL
LIN {X 0,Y 316.993,Z 450.842,A -85,B 0,C 180,E1 15143.932,E2 15143.932} C_VEL
LIN {X 0,Y 315.649,Z 458.412,A -85,B 0,C 180,E1 15143.733,E2 15143.733} C_VEL
LIN {X 0,Y 308.623,Z 478.381,A -85,B 0,C 180,E1 15143.385,E2 15143.385} C_VEL
LIN {X 0,Y 307.604,Z 484.884,A -85,B 0,C 180,E1 15143.198,E2 15143.198} C_VEL
LIN {X 0,Y 305.327,Z 535.75,A -85,B 0,C 180,E1 15141.337,E2 15141.337} C_VEL
LIN {X 0,Y 304.434,Z 552.859,A -85,B 0,C 180,E1 15140.37,E2 15140.37} C_VEL
LIN {X 0,Y 303.412,Z 568.816,A -85,B 0,C 180,E1 15139.137,E2 15139.137} C_VEL
LIN {X 0,Y 302.164,Z 585.322,A -85,B 0,C 180,E1 15137.465,E2 15137.465} C_VEL
LIN {X 0,Y 301.016,Z 599.904,A -85,B 0,C 180,E1 15135.573,E2 15135.573} C_VEL
LIN {X 0,Y 299.896,Z 613.803,A -85,B 0,C 180,E1 15133.297,E2 15133.297} C_VEL
LIN {X 0,Y 299.057,Z 625.03,A -85,B 0,C 180,E1 15130.983,E2 15130.983} C_VEL
LIN {X 0,Y 298.468,Z 634.774,A -85,B 0,C 180,E1 15128.473,E2 15128.473} C_VEL
LIN {X 0,Y 298.151,Z 642.907,A -85,B 0,C 180,E1 15125.771,E2 15125.771} C_VEL
LIN {X 0,Y 298.124,Z 648.944,A -85,B 0,C 180,E1 15123.073,E2 15123.073} C_VEL
LIN {X 0,Y 298.394,Z 653.248,A -85,B 0,C 180,E1 15120.381,E2 15120.381} C_VEL
LIN {X 0,Y 299.003,Z 655.906,A -85,B 0,C 180,E1 15117.506,E2 15117.506} C_VEL
LIN {X 0,Y 300.013,Z 656.757,A -85,B 0,C 180,E1 15114.643,E2 15114.643} C_VEL
LIN {X 0,Y 301.452,Z 655.677,A -85,B 0,C 180,E1 15111.798,E2 15111.798} C_VEL
LIN {X 0,Y 303.402,Z 652.802,A -85,B 0,C 180,E1 15108.978,E2 15108.978} C_VEL
LIN {X 0,Y 306.064,Z 647.539,A -85,B 0,C 180,E1 15106.008,E2 15106.008} C_VEL
LIN {X 0,Y 308.918,Z 640.974,A -85,B 0,C 180,E1 15103.449,E2 15103.449} C_VEL
LIN {X 0,Y 312.297,Z 632.431,A -85,B 0,C 180,E1 15100.937,E2 15100.937} C_VEL
LIN {X 0,Y 315.866,Z 622.296,A -85,B 0,C 180,E1 15098.65,E2 15098.65} C_VEL
LIN {X 0,Y 319.754,Z 610.33,A -85,B 0,C 180,E1 15096.502,E2 15096.502} C_VEL
LIN {X 0,Y 323.96,Z 596.138,A -85,B 0,C 180,E1 15094.496,E2 15094.496} C_VEL
LIN {X 0,Y 328.201,Z 579.971,A -85,B 0,C 180,E1 15092.708,E2 15092.708} C_VEL
LIN {X 0,Y 331.999,Z 563.257,A -85,B 0,C 180,E1 15091.289,E2 15091.289} C_VEL
LIN {X 0,Y 335.343,Z 545.743,A -85,B 0,C 180,E1 15090.172,E2 15090.172} C_VEL
LIN {X 0,Y 346.836,Z 485.385,A -85,B 0,C 180,E1 15087.352,E2 15087.352} C_VEL
LIN {X 0,Y 352.395,Z 457.921,A -85,B 0,C 180,E1 15086.125,E2 15086.125} C_VEL
LIN {X 0,Y 353.575,Z 443.639,A -85,B 0,C 180,E1 15084.501,E2 15084.501} C_VEL
LIN {X 0,Y 355.12,Z 428.655,A -85,B 0,C 180,E1 15082.389,E2 15082.389} C_VEL
LIN {X 0,Y 356.266,Z 420.642,A -85,B 0,C 180,E1 15081.025,E2 15081.025} C_VEL
LIN {X 0,Y 356.445,Z 418.22,A -85,B 0,C 180,E1 15079.186,E2 15079.186} C_VEL
LIN {X 0,Y 357.365,Z 417.577,A -85,B 0,C 180,E1 15077.143,E2 15077.143} C_VEL
LIN {X 0,Y 359.015,Z 419.666,A -85,B 0,C 180,E1 15075.064,E2 15075.064} C_VEL
LIN {X 0,Y 357.648,Z 431.669,A -85,B 0,C 180,E1 15074.006,E2 15074.006} C_VEL
LIN {X 0,Y 345.048,Z 502.692,A -85,B 0,C 180,E1 15071.443,E2 15071.443} C_VEL
LIN {X 0,Y 334.187,Z 577.502,A -85,B 0,C 180,E1 15068.72,E2 15068.72} C_VEL
LIN {X 0,Y 330.227,Z 597.093,A -85,B 0,C 180,E1 15067.708,E2 15067.708} C_VEL
LIN {X 0,Y 325.537,Z 616.491,A -85,B 0,C 180,E1 15066.356,E2 15066.356} C_VEL
LIN {X 0,Y 320.646,Z 634.458,A -85,B 0,C 180,E1 15064.688,E2 15064.688} C_VEL
LIN {X 0,Y 315.723,Z 651.406,A -85,B 0,C 180,E1 15062.682,E2 15062.682} C_VEL
LIN {X 0,Y 311.12,Z 666.81,A -85,B 0,C 180,E1 15060.41,E2 15060.41} C_VEL
LIN {X 0,Y 306.792,Z 681.237,A -85,B 0,C 180,E1 15057.779,E2 15057.779} C_VEL
LIN {X 0,Y 302.991,Z 694.561,A -85,B 0,C 180,E1 15054.779,E2 15054.779} C_VEL
LIN {X 0,Y 300.016,Z 706.347,A -85,B 0,C 180,E1 15051.507,E2 15051.507} C_VEL
LIN {X 0,Y 298.033,Z 716.02,A -85,B 0,C 180,E1 15048.181,E2 15048.181} C_VEL
LIN {X 0,Y 296.946,Z 724.218,A -85,B 0,C 180,E1 15044.629,E2 15044.629} C_VEL
LIN {X 0,Y 296.699,Z 730.435,A -85,B 0,C 180,E1 15041.076,E2 15041.076} C_VEL
LIN {X 0,Y 297.052,Z 734.61,A -85,B 0,C 180,E1 15037.739,E2 15037.739} C_VEL
LIN {X 0,Y 297.663,Z 737.12,A -85,B 0,C 180,E1 15034.432,E2 15034.432} C_VEL
LIN {X 0,Y 298.151,Z 737.885,A -85,B 0,C 180,E1 15031.347,E2 15031.347} C_VEL
LIN {X 0,Y 298.255,Z 737.105,A -85,B 0,C 180,E1 15028.465,E2 15028.465} C_VEL
LIN {X 0,Y 297.994,Z 734.857,A -85,B 0,C 180,E1 15025.575,E2 15025.575} C_VEL
LIN {X 0,Y 297.562,Z 730.709,A -85,B 0,C 180,E1 15022.425,E2 15022.425} C_VEL
LIN {X 0,Y 297.254,Z 724.532,A -85,B 0,C 180,E1 15019.177,E2 15019.177} C_VEL
LIN {X 0,Y 297.321,Z 717.043,A -85,B 0,C 180,E1 15016.188,E2 15016.188} C_VEL
LIN {X 0,Y 297.826,Z 707.692,A -85,B 0,C 180,E1 15013.22,E2 15013.22} C_VEL
LIN {X 0,Y 298.815,Z 696.952,A -85,B 0,C 180,E1 15010.453,E2 15010.453} C_VEL
LIN {X 0,Y 300.276,Z 684.254,A -85,B 0,C 180,E1 15007.776,E2 15007.776} C_VEL
LIN {X 0,Y 302.088,Z 670.147,A -85,B 0,C 180,E1 15005.354,E2 15005.354} C_VEL
LIN {X 0,Y 304.213,Z 654.24,A -85,B 0,C 180,E1 15003.135,E2 15003.135} C_VEL
LIN {X 0,Y 306.294,Z 638.134,A -85,B 0,C 180,E1 15001.325,E2 15001.325} C_VEL
LIN {X 0,Y 308.298,Z 621.32,A -85,B 0,C 180,E1 14999.824,E2 14999.824} C_VEL
LIN {X 0,Y 310.183,Z 603.048,A -85,B 0,C 180,E1 14998.583,E2 14998.583} C_VEL
LIN {X 0,Y 311.694,Z 584.188,A -85,B 0,C 180,E1 14997.671,E2 14997.671} C_VEL
LIN {X 0,Y 312.888,Z 556.668,A -85,B 0,C 180,E1 14996.82,E2 14996.82} C_VEL
LIN {X 0,Y 318.708,Z 420.743,A -85,B 0,C 180,E1 14992.959,E2 14992.959} C_VEL
LIN {X 0,Y 316.556,Z 389.998,A -85,B 0,C 180,E1 14991.799,E2 14991.799} C_VEL
LIN {X 0,Y 319.12,Z 375.603,A -85,B 0,C 180,E1 14989.865,E2 14989.865} C_VEL
LIN {X 0,Y 311.722,Z 352.742,A -85,B 0,C 180,E1 14985.537,E2 14985.537} C_VEL
LIN {X 0,Y 305.44,Z 334.154,A -85,B 0,C 180,E1 14981.648,E2 14981.648} C_VEL
LIN {X 0,Y 299.331,Z 316.77,A -85,B 0,C 180,E1 14977.663,E2 14977.663} C_VEL
LIN {X 0,Y 298.229,Z 313.65,A -85,B 0,C 180,E1 14976.881,E2 14976.881} C_VEL
LIN {X 0,Y 298.242,Z 313.648,A -85,B 0,C 180,E1 14972.214,E2 14972.214} C_VEL
LIN {X 0,Y 298.27,Z 313.647,A -85,B 0,C 180,E1 14967.755,E2 14967.755} C_VEL
LIN {X 0,Y 298.241,Z 313.648,A -85,B 0,C 180,E1 14963.097,E2 14963.097} C_VEL
LIN {X 0,Y 298.237,Z 313.647,A -85,B 0,C 180,E1 14958.424,E2 14958.424} C_VEL
LIN {X 0,Y 298.253,Z 313.646,A -85,B 0,C 180,E1 14953.97,E2 14953.97} C_VEL
LIN {X 0,Y 298.262,Z 313.642,A -85,B 0,C 180,E1 14949.457,E2 14949.457} C_VEL
LIN {X 0,Y 298.243,Z 313.645,A -85,B 0,C 180,E1 14945.003,E2 14945.003} C_VEL
LIN {X 0,Y 298.238,Z 313.646,A -85,B 0,C 180,E1 14940.387,E2 14940.387} C_VEL
LIN {X 0,Y 298.26,Z 313.643,A -85,B 0,C 180,E1 14935.773,E2 14935.773} C_VEL
LIN {X 0,Y 298.268,Z 313.64,A -85,B 0,C 180,E1 14931.327,E2 14931.327} C_VEL
LIN {X 0,Y 298.246,Z 313.644,A -85,B 0,C 180,E1 14926.826,E2 14926.826} C_VEL
LIN {X 0,Y 298.247,Z 313.642,A -85,B 0,C 180,E1 14922.188,E2 14922.188} C_VEL
LIN {X 0,Y 298.285,Z 313.643,A -85,B 0,C 180,E1 14917.538,E2 14917.538} C_VEL
LIN {X 0,Y 298.254,Z 313.64,A -85,B 0,C 180,E1 14912.879,E2 14912.879} C_VEL
LIN {X 0,Y 298.248,Z 313.64,A -85,B 0,C 180,E1 14908.246,E2 14908.246} C_VEL
LIN {X 0,Y 298.271,Z 313.645,A -85,B 0,C 180,E1 14903.61,E2 14903.61} C_VEL
LIN {X 0,Y 298.277,Z 313.633,A -85,B 0,C 180,E1 14899.186,E2 14899.186} C_VEL
LIN {X 0,Y 298.256,Z 313.642,A -85,B 0,C 180,E1 14894.713,E2 14894.713} C_VEL
LIN {X 0,Y 298.255,Z 313.642,A -85,B 0,C 180,E1 14890.063,E2 14890.063} C_VEL
LIN {X 0,Y 298.275,Z 313.636,A -85,B 0,C 180,E1 14885.462,E2 14885.462} C_VEL
LIN {X 0,Y 298.267,Z 313.642,A -85,B 0,C 180,E1 14880.896,E2 14880.896} C_VEL
LIN {X 0,Y 298.257,Z 313.638,A -85,B 0,C 180,E1 14876.477,E2 14876.477} C_VEL
LIN {X 0,Y 298.261,Z 313.64,A -85,B 0,C 180,E1 14871.844,E2 14871.844} C_VEL
LIN {X 0,Y 298.282,Z 313.642,A -85,B 0,C 180,E1 14867.356,E2 14867.356} C_VEL
LIN {X 0,Y 298.277,Z 313.637,A -85,B 0,C 180,E1 14862.977,E2 14862.977} C_VEL
LIN {X 0,Y 298.259,Z 313.643,A -85,B 0,C 180,E1 14858.481,E2 14858.481} C_VEL
LIN {X 0,Y 298.262,Z 313.638,A -85,B 0,C 180,E1 14853.843,E2 14853.843} C_VEL
LIN {X 0,Y 298.294,Z 313.641,A -85,B 0,C 180,E1 14849.23,E2 14849.23} C_VEL
LIN {X 0,Y 298.268,Z 313.64,A -85,B 0,C 180,E1 14844.585,E2 14844.585} C_VEL
LIN {X 0,Y 298.263,Z 313.641,A -85,B 0,C 180,E1 14839.96,E2 14839.96} C_VEL
LIN {X 0,Y 298.284,Z 313.644,A -85,B 0,C 180,E1 14835.438,E2 14835.438} C_VEL
LIN {X 0,Y 298.284,Z 313.64,A -85,B 0,C 180,E1 14830.821,E2 14830.821} C_VEL
LIN {X 0,Y 298.267,Z 313.642,A -85,B 0,C 180,E1 14826.218,E2 14826.218} C_VEL
LIN {X 0,Y 298.281,Z 313.644,A -85,B 0,C 180,E1 14821.574,E2 14821.574} C_VEL
LIN {X 0,Y 298.295,Z 313.642,A -85,B 0,C 180,E1 14817.11,E2 14817.11} C_VEL
LIN {X 0,Y 298.282,Z 313.642,A -85,B 0,C 180,E1 14812.596,E2 14812.596} C_VEL
LIN {X 0,Y 298.27,Z 313.645,A -85,B 0,C 180,E1 14808.084,E2 14808.084} C_VEL
LIN {X 0,Y 298.288,Z 313.689,A -85,B 0,C 180,E1 14805.463,E2 14805.463} C_VEL
LIN {X 0,Y 303.11,Z 329.98,A -85,B 0,C 180,E1 14801.226,E2 14801.226} C_VEL
LIN {X 0,Y 307.685,Z 346.67,A -85,B 0,C 180,E1 14797.183,E2 14797.183} C_VEL
LIN {X 0,Y 311.657,Z 362.758,A -85,B 0,C 180,E1 14793.542,E2 14793.542} C_VEL
LIN {X 0,Y 307.736,Z 389.159,A -85,B 0,C 180,E1 14788.685,E2 14788.685} C_VEL
LIN {X 0,Y 306.181,Z 401.425,A -85,B 0,C 180,E1 14786.499,E2 14786.499} C_VEL
LIN {X 0,Y 309.977,Z 439.747,A -85,B 0,C 180,E1 14784.769,E2 14784.769} C_VEL
LIN {X 0,Y 307.604,Z 484.884,A -85,B 0,C 180,E1 14783.198,E2 14783.198} C_VEL
LIN {X 0,Y 306.283,Z 492.451,A -85,B 0,C 180,E1 14782.985,E2 14782.985} C_VEL
LIN {X 0,Y 299.244,Z 512.388,A -85,B 0,C 180,E1 14782.574,E2 14782.574} C_VEL
LIN {X 0,Y 298.239,Z 518.883,A -85,B 0,C 180,E1 14782.37,E2 14782.37} C_VEL
LIN {X 0,Y 297.299,Z 540.775,A -85,B 0,C 180,E1 14781.437,E2 14781.437} C_VEL
LIN {X 0,Y 296.305,Z 558.122,A -85,B 0,C 180,E1 14780.335,E2 14780.335} C_VEL
LIN {X 0,Y 295.103,Z 575.357,A -85,B 0,C 180,E1 14778.841,E2 14778.841} C_VEL
LIN {X 0,Y 293.828,Z 591.498,A -85,B 0,C 180,E1 14777.013,E2 14777.013} C_VEL
LIN {X 0,Y 292.652,Z 605.863,A -85,B 0,C 180,E1 14774.945,E2 14774.945} C_VEL
LIN {X 0,Y 291.6,Z 618.919,A -85,B 0,C 180,E1 14772.573,E2 14772.573} C_VEL
LIN {X 0,Y 290.822,Z 629.742,A -85,B 0,C 180,E1 14770.095,E2 14770.095} C_VEL
LIN {X 0,Y 290.341,Z 638.751,A -85,B 0,C 180,E1 14767.516,E2 14767.516} C_VEL
LIN {X 0,Y 290.141,Z 646.254,A -85,B 0,C 180,E1 14764.741,E2 14764.741} C_VEL
LIN {X 0,Y 290.247,Z 651.783,A -85,B 0,C 180,E1 14761.971,E2 14761.971} C_VEL
LIN {X 0,Y 290.703,Z 655.775,A -85,B 0,C 180,E1 14759.012,E2 14759.012} C_VEL
LIN {X 0,Y 291.543,Z 657.832,A -85,B 0,C 180,E1 14756.064,E2 14756.064} C_VEL
LIN {X 0,Y 292.846,Z 658.087,A -85,B 0,C 180,E1 14753.134,E2 14753.134} C_VEL
LIN {X 0,Y 294.629,Z 656.442,A -85,B 0,C 180,E1 14750.228,E2 14750.228} C_VEL
LIN {X 0,Y 296.981,Z 653.001,A -85,B 0,C 180,E1 14747.357,E2 14747.357} C_VEL
LIN {X 0,Y 299.681,Z 647.965,A -85,B 0,C 180,E1 14744.715,E2 14744.715} C_VEL
LIN {X 0,Y 302.929,Z 641.179,A -85,B 0,C 180,E1 14742.122,E2 14742.122} C_VEL
LIN {X 0,Y 306.688,Z 632.289,A -85,B 0,C 180,E1 14739.581,E2 14739.581} C_VEL
LIN {X 0,Y 310.68,Z 622.005,A -85,B 0,C 180,E1 14737.28,E2 14737.28} C_VEL
LIN {X 0,Y 315.354,Z 608.72,A -85,B 0,C 180,E1 14734.956,E2 14734.956} C_VEL
LIN {X 0,Y 320.004,Z 594.035,A -85,B 0,C 180,E1 14732.957,E2 14732.957} C_VEL
LIN {X 0,Y 324.458,Z 578.154,A -85,B 0,C 180,E1 14731.265,E2 14731.265} C_VEL
LIN {X 0,Y 328.383,Z 562.08,A -85,B 0,C 180,E1 14729.94,E2 14729.94} C_VEL
LIN {X 0,Y 332.042,Z 544.127,A -85,B 0,C 180,E1 14728.829,E2 14728.829} C_VEL
LIN {X 0,Y 349.433,Z 460.631,A -85,B 0,C 180,E1 14724.979,E2 14724.979} C_VEL
LIN {X 0,Y 351.189,Z 445.711,A -85,B 0,C 180,E1 14723.203,E2 14723.203} C_VEL
LIN {X 0,Y 353.387,Z 431.475,A -85,B 0,C 180,E1 14721.086,E2 14721.086} C_VEL
LIN {X 0,Y 354.129,Z 427.63,A -85,B 0,C 180,E1 14720.427,E2 14720.427} C_VEL
LIN {X 0,Y 354.594,Z 425.556,A -85,B 0,C 180,E1 14718.596,E2 14718.596} C_VEL
LIN {X 0,Y 355.597,Z 425.566,A -85,B 0,C 180,E1 14716.741,E2 14716.741} C_VEL
LIN {X 0,Y 356.242,Z 426.745,A -85,B 0,C 180,E1 14715.803,E2 14715.803} C_VEL
LIN {X 0,Y 355.042,Z 434.634,A -85,B 0,C 180,E1 14715.16,E2 14715.16} C_VEL
LIN {X 0,Y 341.314,Z 505.731,A -85,B 0,C 180,E1 14712.566,E2 14712.566} C_VEL
LIN {X 0,Y 329.937,Z 576.623,A -85,B 0,C 180,E1 14709.92,E2 14709.92} C_VEL
LIN {X 0,Y 325.354,Z 597.309,A -85,B 0,C 180,E1 14708.825,E2 14708.825} C_VEL
LIN {X 0,Y 320.396,Z 616.032,A -85,B 0,C 180,E1 14707.485,E2 14707.485} C_VEL
LIN {X 0,Y 315.256,Z 633.376,A -85,B 0,C 180,E1 14705.845,E2 14705.845} C_VEL
LIN {X 0,Y 309.988,Z 650.069,A -85,B 0,C 180,E1 14703.841,E2 14703.841} C_VEL
LIN {X 0,Y 304.791,Z 665.991,A -85,B 0,C 180,E1 14701.441,E2 14701.441} C_VEL
LIN {X 0,Y 299.957,Z 680.599,A -85,B 0,C 180,E1 14698.687,E2 14698.687} C_VEL
LIN {X 0,Y 295.834,Z 693.712,A -85,B 0,C 180,E1 14695.635,E2 14695.635} C_VEL
LIN {X 0,Y 292.564,Z 705.331,A -85,B 0,C 180,E1 14692.295,E2 14692.295} C_VEL
LIN {X 0,Y 290.339,Z 714.878,A -85,B 0,C 180,E1 14688.889,E2 14688.889} C_VEL
LIN {X 0,Y 289.05,Z 723.073,A -85,B 0,C 180,E1 14685.177,E2 14685.177} C_VEL
LIN {X 0,Y 288.708,Z 729.312,A -85,B 0,C 180,E1 14681.445,E2 14681.445} C_VEL
LIN {X 0,Y 289.065,Z 733.439,A -85,B 0,C 180,E1 14677.954,E2 14677.954} C_VEL
LIN {X 0,Y 289.72,Z 735.835,A -85,B 0,C 180,E1 14674.554,E2 14674.554} C_VEL
LIN {X 0,Y 290.235,Z 736.537,A -85,B 0,C 180,E1 14671.581,E2 14671.581} C_VEL
LIN {X 0,Y 290.396,Z 735.83,A -85,B 0,C 180,E1 14668.818,E2 14668.818} C_VEL
LIN {X 0,Y 290.161,Z 733.649,A -85,B 0,C 180,E1 14665.852,E2 14665.852} C_VEL
LIN {X 0,Y 289.703,Z 729.623,A -85,B 0,C 180,E1 14662.665,E2 14662.665} C_VEL
LIN {X 0,Y 289.36,Z 723.76,A -85,B 0,C 180,E1 14659.449,E2 14659.449} C_VEL
LIN {X 0,Y 289.394,Z 715.929,A -85,B 0,C 180,E1 14656.21,E2 14656.21} C_VEL
LIN {X 0,Y 289.893,Z 706.579,A -85,B 0,C 180,E1 14653.16,E2 14653.16} C_VEL
LIN {X 0,Y 290.893,Z 695.826,A -85,B 0,C 180,E1 14650.317,E2 14650.317} C_VEL
LIN {X 0,Y 292.381,Z 683.113,A -85,B 0,C 180,E1 14647.572,E2 14647.572} C_VEL
LIN {X 0,Y 294.245,Z 668.933,A -85,B 0,C 180,E1 14645.081,E2 14645.081} C_VEL
LIN {X 0,Y 296.423,Z 652.967,A -85,B 0,C 180,E1 14642.805,E2 14642.805} C_VEL
LIN {X 0,Y 298.582,Z 636.607,A -85,B 0,C 180,E1 14640.931,E2 14640.931} C_VEL
LIN {X 0,Y 300.615,Z 619.864,A -85,B 0,C 180,E1 14639.412,E2 14639.412} C_VEL
LIN {X 0,Y 302.584,Z 601.132,A -85,B 0,C 180,E1 14638.131,E2 14638.131} C_VEL
LIN {X 0,Y 304.121,Z 581.604,A -85,B 0,C 180,E1 14637.185,E2 14637.185} C_VEL
LIN {X 0,Y 305.909,Z 539.567,A -85,B 0,C 180,E1 14635.905,E2 14635.905} C_VEL
LIN {X 0,Y 311.281,Z 421.492,A -85,B 0,C 180,E1 14632.427,E2 14632.427} C_VEL
LIN {X 0,Y 309.206,Z 390.001,A -85,B 0,C 180,E1 14631.2,E2 14631.2} C_VEL
LIN {X 0,Y 311.523,Z 377.833,A -85,B 0,C 180,E1 14629.526,E2 14629.526} C_VEL
LIN {X 0,Y 304.368,Z 355.498,A -85,B 0,C 180,E1 14625.202,E2 14625.202} C_VEL
LIN {X 0,Y 297.928,Z 336.524,A -85,B 0,C 180,E1 14621.134,E2 14621.134} C_VEL
LIN {X 0,Y 292.16,Z 320.171,A -85,B 0,C 180,E1 14617.285,E2 14617.285} C_VEL
LIN {X 0,Y 290.314,Z 314.634,A -85,B 0,C 180,E1 14615.84,E2 14615.84} C_VEL
LIN {X 0,Y 290.312,Z 314.634,A -85,B 0,C 180,E1 14611.339,E2 14611.339} C_VEL
LIN {X 0,Y 290.294,Z 314.634,A -85,B 0,C 180,E1 14606.823,E2 14606.823} C_VEL
LIN {X 0,Y 290.308,Z 314.637,A -85,B 0,C 180,E1 14602.113,E2 14602.113} C_VEL
LIN {X 0,Y 290.32,Z 314.633,A -85,B 0,C 180,E1 14597.455,E2 14597.455} C_VEL
LIN {X 0,Y 290.299,Z 314.633,A -85,B 0,C 180,E1 14592.919,E2 14592.919} C_VEL
LIN {X 0,Y 290.299,Z 314.631,A -85,B 0,C 180,E1 14588.32,E2 14588.32} C_VEL
LIN {X 0,Y 290.319,Z 314.633,A -85,B 0,C 180,E1 14583.755,E2 14583.755} C_VEL
LIN {X 0,Y 290.318,Z 314.632,A -85,B 0,C 180,E1 14579.214,E2 14579.214} C_VEL
LIN {X 0,Y 290.299,Z 314.634,A -85,B 0,C 180,E1 14574.469,E2 14574.469} C_VEL
LIN {X 0,Y 290.317,Z 314.63,A -85,B 0,C 180,E1 14569.887,E2 14569.887} C_VEL
LIN {X 0,Y 290.327,Z 314.633,A -85,B 0,C 180,E1 14565.239,E2 14565.239} C_VEL
LIN {X 0,Y 290.306,Z 314.625,A -85,B 0,C 180,E1 14560.677,E2 14560.677} C_VEL
LIN {X 0,Y 290.316,Z 314.634,A -85,B 0,C 180,E1 14556.025,E2 14556.025} C_VEL
LIN {X 0,Y 290.344,Z 314.621,A -85,B 0,C 180,E1 14551.405,E2 14551.405} C_VEL
LIN {X 0,Y 290.316,Z 314.631,A -85,B 0,C 180,E1 14546.802,E2 14546.802} C_VEL
LIN {X 0,Y 290.315,Z 314.631,A -85,B 0,C 180,E1 14542.06,E2 14542.06} C_VEL
LIN {X 0,Y 290.337,Z 314.624,A -85,B 0,C 180,E1 14537.471,E2 14537.471} C_VEL
LIN {X 0,Y 290.32,Z 314.631,A -85,B 0,C 180,E1 14532.819,E2 14532.819} C_VEL
LIN {X 0,Y 290.316,Z 314.626,A -85,B 0,C 180,E1 14528.058,E2 14528.058} C_VEL
LIN {X 0,Y 290.343,Z 314.629,A -85,B 0,C 180,E1 14523.433,E2 14523.433} C_VEL
LIN {X 0,Y 290.328,Z 314.629,A -85,B 0,C 180,E1 14518.824,E2 14518.824} C_VEL
LIN {X 0,Y 290.318,Z 314.621,A -85,B 0,C 180,E1 14514.134,E2 14514.134} C_VEL
LIN {X 0,Y 290.339,Z 314.633,A -85,B 0,C 180,E1 14509.513,E2 14509.513} C_VEL
LIN {X 0,Y 290.338,Z 314.624,A -85,B 0,C 180,E1 14504.967,E2 14504.967} C_VEL
LIN {X 0,Y 290.319,Z 314.63,A -85,B 0,C 180,E1 14500.315,E2 14500.315} C_VEL
LIN {X 0,Y 290.329,Z 314.631,A -85,B 0,C 180,E1 14495.73,E2 14495.73} C_VEL
LIN {X 0,Y 290.351,Z 314.631,A -85,B 0,C 180,E1 14491.182,E2 14491.182} C_VEL
LIN {X 0,Y 290.329,Z 314.625,A -85,B 0,C 180,E1 14486.642,E2 14486.642} C_VEL
LIN {X 0,Y 290.326,Z 314.632,A -85,B 0,C 180,E1 14481.881,E2 14481.881} C_VEL
LIN {X 0,Y 290.349,Z 314.632,A -85,B 0,C 180,E1 14477.266,E2 14477.266} C_VEL
LIN {X 0,Y 290.341,Z 314.629,A -85,B 0,C 180,E1 14472.771,E2 14472.771} C_VEL
LIN {X 0,Y 290.326,Z 314.63,A -85,B 0,C 180,E1 14468.163,E2 14468.163} C_VEL
LIN {X 0,Y 290.341,Z 314.633,A -85,B 0,C 180,E1 14463.547,E2 14463.547} C_VEL
LIN {X 0,Y 290.361,Z 314.628,A -85,B 0,C 180,E1 14459.022,E2 14459.022} C_VEL
LIN {X 0,Y 290.333,Z 314.631,A -85,B 0,C 180,E1 14454.358,E2 14454.358} C_VEL
LIN {X 0,Y 290.336,Z 314.635,A -85,B 0,C 180,E1 14449.65,E2 14449.65} C_VEL
LIN {X 0,Y 290.354,Z 314.766,A -85,B 0,C 180,E1 14446.31,E2 14446.31} C_VEL
LIN {X 0,Y 295.204,Z 330.913,A -85,B 0,C 180,E1 14441.972,E2 14441.972} C_VEL
LIN {X 0,Y 299.801,Z 347.796,A -85,B 0,C 180,E1 14437.774,E2 14437.774} C_VEL
LIN {X 0,Y 303.953,Z 364.532,A -85,B 0,C 180,E1 14433.884,E2 14433.884} C_VEL
LIN {X 0,Y 300.189,Z 389.309,A -85,B 0,C 180,E1 14429.228,E2 14429.228} C_VEL
LIN {X 0,Y 298.594,Z 401.239,A -85,B 0,C 180,E1 14427.051,E2 14427.051} C_VEL
LIN {X 0,Y 302.366,Z 440.537,A -85,B 0,C 180,E1 14425.227,E2 14425.227} C_VEL
LIN {X 0,Y 298.239,Z 518.883,A -85,B 0,C 180,E1 14422.37,E2 14422.37} C_VEL
LIN {X 0,Y 296.971,Z 526.451,A -85,B 0,C 180,E1 14422.13,E2 14422.13} C_VEL
LIN {X 0,Y 290.267,Z 545.177,A -85,B 0,C 180,E1 14421.52,E2 14421.52} C_VEL
LIN {X 0,Y 288.863,Z 552.489,A -85,B 0,C 180,E1 14421.091,E2 14421.091} C_VEL
LIN {X 0,Y 287.694,Z 569.915,A -85,B 0,C 180,E1 14419.698,E2 14419.698} C_VEL
LIN {X 0,Y 286.41,Z 586.058,A -85,B 0,C 180,E1 14417.993,E2 14417.993} C_VEL
LIN {X 0,Y 285.115,Z 601.692,A -85,B 0,C 180,E1 14415.871,E2 14415.871} C_VEL
LIN {X 0,Y 283.93,Z 615.831,A -85,B 0,C 180,E1 14413.436,E2 14413.436} C_VEL
LIN {X 0,Y 283.029,Z 627.71,A -85,B 0,C 180,E1 14410.852,E2 14410.852} C_VEL
LIN {X 0,Y 282.478,Z 636.955,A -85,B 0,C 180,E1 14408.341,E2 14408.341} C_VEL
LIN {X 0,Y 282.193,Z 645.236,A -85,B 0,C 180,E1 14405.487,E2 14405.487} C_VEL
LIN {X 0,Y 282.238,Z 651.618,A -85,B 0,C 180,E1 14402.515,E2 14402.515} C_VEL
LIN {X 0,Y 282.64,Z 656.075,A -85,B 0,C 180,E1 14399.592,E2 14399.592} C_VEL
LIN {X 0,Y 283.447,Z 658.784,A -85,B 0,C 180,E1 14396.559,E2 14396.559} C_VEL
LIN {X 0,Y 284.638,Z 659.698,A -85,B 0,C 180,E1 14393.746,E2 14393.746} C_VEL
LIN {X 0,Y 286.405,Z 658.85,A -85,B 0,C 180,E1 14390.756,E2 14390.756} C_VEL
LIN {X 0,Y 288.751,Z 656.229,A -85,B 0,C 180,E1 14387.803,E2 14387.803} C_VEL
LIN {X 0,Y 291.702,Z 651.713,A -85,B 0,C 180,E1 14384.898,E2 14384.898} C_VEL
LIN {X 0,Y 295.287,Z 645.217,A -85,B 0,C 180,E1 14382.051,E2 14382.051} C_VEL
LIN {X 0,Y 299.504,Z 636.513,A -85,B 0,C 180,E1 14379.273,E2 14379.273} C_VEL
LIN {X 0,Y 303.689,Z 626.988,A -85,B 0,C 180,E1 14376.932,E2 14376.932} C_VEL
LIN {X 0,Y 308.581,Z 614.808,A -85,B 0,C 180,E1 14374.573,E2 14374.573} C_VEL
LIN {X 0,Y 313.859,Z 600.221,A -85,B 0,C 180,E1 14372.383,E2 14372.383} C_VEL
LIN {X 0,Y 318.981,Z 584.209,A -85,B 0,C 180,E1 14370.518,E2 14370.518} C_VEL
LIN {X 0,Y 323.592,Z 567.678,A -85,B 0,C 180,E1 14369.036,E2 14369.036} C_VEL
LIN {X 0,Y 327.624,Z 550.479,A -85,B 0,C 180,E1 14367.872,E2 14367.872} C_VEL
LIN {X 0,Y 337.315,Z 505.287,A -85,B 0,C 180,E1 14365.67,E2 14365.67} C_VEL
LIN {X 0,Y 346.9,Z 463.227,A -85,B 0,C 180,E1 14363.78,E2 14363.78} C_VEL
LIN {X 0,Y 349.143,Z 448.862,A -85,B 0,C 180,E1 14361.995,E2 14361.995} C_VEL
LIN {X 0,Y 351.697,Z 436.331,A -85,B 0,C 180,E1 14360.077,E2 14360.077} C_VEL
LIN {X 0,Y 352.123,Z 434.582,A -85,B 0,C 180,E1 14359.758,E2 14359.758} C_VEL
LIN {X 0,Y 352.716,Z 433.199,A -85,B 0,C 180,E1 14358.207,E2 14358.207} C_VEL
LIN {X 0,Y 353.545,Z 433.311,A -85,B 0,C 180,E1 14356.81,E2 14356.81} C_VEL
LIN {X 0,Y 353.643,Z 433.648,A -85,B 0,C 180,E1 14356.602,E2 14356.602} C_VEL
LIN {X 0,Y 352.888,Z 437.366,A -85,B 0,C 180,E1 14356.351,E2 14356.351} C_VEL
LIN {X 0,Y 337.771,Z 509.632,A -85,B 0,C 180,E1 14353.697,E2 14353.697} C_VEL
LIN {X 0,Y 326.265,Z 574.885,A -85,B 0,C 180,E1 14351.216,E2 14351.216} C_VEL
LIN {X 0,Y 321.568,Z 594.623,A -85,B 0,C 180,E1 14350.181,E2 14350.181} C_VEL
LIN {X 0,Y 316.287,Z 613.287,A -85,B 0,C 180,E1 14348.868,E2 14348.868} C_VEL
LIN {X 0,Y 310.677,Z 630.848,A -85,B 0,C 180,E1 14347.234,E2 14347.234} C_VEL
LIN {X 0,Y 304.755,Z 648.12,A -85,B 0,C 180,E1 14345.157,E2 14345.157} C_VEL
LIN {X 0,Y 299.162,Z 663.786,A -85,B 0,C 180,E1 14342.783,E2 14342.783} C_VEL
LIN {X 0,Y 293.868,Z 678.38,A -85,B 0,C 180,E1 14340.012,E2 14340.012} C_VEL
LIN {X 0,Y 289.198,Z 691.689,A -85,B 0,C 180,E1 14336.871,E2 14336.871} C_VEL
LIN {X 0,Y 285.419,Z 703.587,A -85,B 0,C 180,E1 14333.386,E2 14333.386} C_VEL
LIN {X 0,Y 282.81,Z 713.278,A -85,B 0,C 180,E1 14329.842,E2 14329.842} C_VEL
LIN {X 0,Y 281.258,Z 721.337,A -85,B 0,C 180,E1 14326.1,E2 14326.1} C_VEL
LIN {X 0,Y 280.722,Z 727.528,A -85,B 0,C 180,E1 14322.341,E2 14322.341} C_VEL
LIN {X 0,Y 281.007,Z 731.909,A -85,B 0,C 180,E1 14318.596,E2 14318.596} C_VEL
LIN {X 0,Y 281.684,Z 734.379,A -85,B 0,C 180,E1 14315.093,E2 14315.093} C_VEL
LIN {X 0,Y 282.286,Z 735.158,A -85,B 0,C 180,E1 14312.031,E2 14312.031} C_VEL
LIN {X 0,Y 282.54,Z 734.524,A -85,B 0,C 180,E1 14309.19,E2 14309.19} C_VEL
LIN {X 0,Y 282.334,Z 732.406,A -85,B 0,C 180,E1 14306.143,E2 14306.143} C_VEL
LIN {X 0,Y 281.848,Z 728.423,A -85,B 0,C 180,E1 14302.869,E2 14302.869} C_VEL
LIN {X 0,Y 281.468,Z 722.583,A -85,B 0,C 180,E1 14299.564,E2 14299.564} C_VEL
LIN {X 0,Y 281.474,Z 714.757,A -85,B 0,C 180,E1 14296.233,E2 14296.233} C_VEL
LIN {X 0,Y 281.965,Z 705.397,A -85,B 0,C 180,E1 14293.097,E2 14293.097} C_VEL
LIN {X 0,Y 282.977,Z 694.62,A -85,B 0,C 180,E1 14290.173,E2 14290.173} C_VEL
LIN {X 0,Y 284.488,Z 681.924,A -85,B 0,C 180,E1 14287.368,E2 14287.368} C_VEL
LIN {X 0,Y 286.412,Z 667.608,A -85,B 0,C 180,E1 14284.794,E2 14284.794} C_VEL
LIN {X 0,Y 288.621,Z 651.764,A -85,B 0,C 180,E1 14282.484,E2 14282.484} C_VEL
LIN {X 0,Y 290.841,Z 635.292,A -85,B 0,C 180,E1 14280.556,E2 14280.556} C_VEL
LIN {X 0,Y 292.95,Z 618.144,A -85,B 0,C 180,E1 14278.98,E2 14278.98} C_VEL
LIN {X 0,Y 294.891,Z 600.142,A -85,B 0,C 180,E1 14277.724,E2 14277.724} C_VEL
LIN {X 0,Y 296.432,Z 580.875,A -85,B 0,C 180,E1 14276.765,E2 14276.765} C_VEL
LIN {X 0,Y 298.693,Z 530.008,A -85,B 0,C 180,E1 14275.167,E2 14275.167} C_VEL
LIN {X 0,Y 303.829,Z 422.107,A -85,B 0,C 180,E1 14271.883,E2 14271.883} C_VEL
LIN {X 0,Y 301.845,Z 390.143,A -85,B 0,C 180,E1 14270.6,E2 14270.6} C_VEL
LIN {X 0,Y 303.907,Z 380.005,A -85,B 0,C 180,E1 14269.177,E2 14269.177} C_VEL
LIN {X 0,Y 296.981,Z 358.202,A -85,B 0,C 180,E1 14264.859,E2 14264.859} C_VEL
LIN {X 0,Y 290.222,Z 338.032,A -85,B 0,C 180,E1 14260.417,E2 14260.417} C_VEL
LIN {X 0,Y 284.114,Z 320.964,A -85,B 0,C 180,E1 14256.247,E2 14256.247} C_VEL
LIN {X 0,Y 282.353,Z 315.628,A -85,B 0,C 180,E1 14254.873,E2 14254.873} C_VEL
LIN {X 0,Y 282.363,Z 315.626,A -85,B 0,C 180,E1 14250.19,E2 14250.19} C_VEL
LIN {X 0,Y 282.381,Z 315.626,A -85,B 0,C 180,E1 14245.596,E2 14245.596} C_VEL
LIN {X 0,Y 282.361,Z 315.623,A -85,B 0,C 180,E1 14240.958,E2 14240.958} C_VEL
LIN {X 0,Y 282.364,Z 315.622,A -85,B 0,C 180,E1 14236.247,E2 14236.247} C_VEL
LIN {X 0,Y 282.383,Z 315.624,A -85,B 0,C 180,E1 14231.646,E2 14231.646} C_VEL
LIN {X 0,Y 282.363,Z 315.624,A -85,B 0,C 180,E1 14226.918,E2 14226.918} C_VEL
LIN {X 0,Y 282.364,Z 315.621,A -85,B 0,C 180,E1 14222.235,E2 14222.235} C_VEL
LIN {X 0,Y 282.382,Z 315.62,A -85,B 0,C 180,E1 14217.771,E2 14217.771} C_VEL
LIN {X 0,Y 282.375,Z 315.622,A -85,B 0,C 180,E1 14213.088,E2 14213.088} C_VEL
LIN {X 0,Y 282.364,Z 315.619,A -85,B 0,C 180,E1 14208.359,E2 14208.359} C_VEL
LIN {X 0,Y 282.386,Z 315.623,A -85,B 0,C 180,E1 14203.76,E2 14203.76} C_VEL
LIN {X 0,Y 282.38,Z 315.619,A -85,B 0,C 180,E1 14199.049,E2 14199.049} C_VEL
LIN {X 0,Y 282.369,Z 315.621,A -85,B 0,C 180,E1 14194.409,E2 14194.409} C_VEL
LIN {X 0,Y 282.388,Z 315.61,A -85,B 0,C 180,E1 14189.758,E2 14189.758} C_VEL
LIN {X 0,Y 282.39,Z 315.621,A -85,B 0,C 180,E1 14185.226,E2 14185.226} C_VEL
LIN {X 0,Y 282.37,Z 315.613,A -85,B 0,C 180,E1 14180.524,E2 14180.524} C_VEL
LIN {X 0,Y 282.386,Z 315.617,A -85,B 0,C 180,E1 14175.776,E2 14175.776} C_VEL
LIN {X 0,Y 282.394,Z 315.617,A -85,B 0,C 180,E1 14171.054,E2 14171.054} C_VEL
LIN {X 0,Y 282.375,Z 315.607,A -85,B 0,C 180,E1 14166.501,E2 14166.501} C_VEL
LIN {X 0,Y 282.388,Z 315.62,A -85,B 0,C 180,E1 14161.821,E2 14161.821} C_VEL
LIN {X 0,Y 282.403,Z 315.614,A -85,B 0,C 180,E1 14157.174,E2 14157.174} C_VEL
LIN {X 0,Y 282.381,Z 315.615,A -85,B 0,C 180,E1 14152.47,E2 14152.47} C_VEL
LIN {X 0,Y 282.393,Z 315.622,A -85,B 0,C 180,E1 14147.726,E2 14147.726} C_VEL
LIN {X 0,Y 282.405,Z 315.612,A -85,B 0,C 180,E1 14143.095,E2 14143.095} C_VEL
LIN {X 0,Y 282.38,Z 315.621,A -85,B 0,C 180,E1 14138.346,E2 14138.346} C_VEL
LIN {X 0,Y 282.391,Z 315.614,A -85,B 0,C 180,E1 14133.653,E2 14133.653} C_VEL
LIN {X 0,Y 282.407,Z 315.618,A -85,B 0,C 180,E1 14128.984,E2 14128.984} C_VEL
LIN {X 0,Y 282.384,Z 315.618,A -85,B 0,C 180,E1 14124.202,E2 14124.202} C_VEL
LIN {X 0,Y 282.396,Z 315.618,A -85,B 0,C 180,E1 14119.595,E2 14119.595} C_VEL
LIN {X 0,Y 282.417,Z 315.616,A -85,B 0,C 180,E1 14115.021,E2 14115.021} C_VEL
LIN {X 0,Y 282.39,Z 315.619,A -85,B 0,C 180,E1 14110.343,E2 14110.343} C_VEL
LIN {X 0,Y 282.394,Z 315.622,A -85,B 0,C 180,E1 14105.749,E2 14105.749} C_VEL
LIN {X 0,Y 282.423,Z 315.618,A -85,B 0,C 180,E1 14100.972,E2 14100.972} C_VEL
LIN {X 0,Y 282.392,Z 315.62,A -85,B 0,C 180,E1 14096.227,E2 14096.227} C_VEL
LIN {X 0,Y 282.407,Z 315.622,A -85,B 0,C 180,E1 14091.453,E2 14091.453} C_VEL
LIN {X 0,Y 282.413,Z 315.623,A -85,B 0,C 180,E1 14087.248,E2 14087.248} C_VEL
LIN {X 0,Y 287.387,Z 332.298,A -85,B 0,C 180,E1 14082.635,E2 14082.635} C_VEL
LIN {X 0,Y 291.836,Z 348.487,A -85,B 0,C 180,E1 14078.49,E2 14078.49} C_VEL
LIN {X 0,Y 296.151,Z 365.964,A -85,B 0,C 180,E1 14074.316,E2 14074.316} C_VEL
LIN {X 0,Y 296.033,Z 368.458,A -85,B 0,C 180,E1 14073.809,E2 14073.809} C_VEL
LIN {X 0,Y 291.677,Z 395.857,A -85,B 0,C 180,E1 14068.564,E2 14068.564} C_VEL
LIN {X 0,Y 291.003,Z 401.157,A -85,B 0,C 180,E1 14067.6,E2 14067.6} C_VEL
LIN {X 0,Y 294.724,Z 441.27,A -85,B 0,C 180,E1 14065.679,E2 14065.679} C_VEL
LIN {X 0,Y 289.738,Z 536.406,A -85,B 0,C 180,E1 14062.025,E2 14062.025} C_VEL
LIN {X 0,Y 288.863,Z 552.489,A -85,B 0,C 180,E1 14061.091,E2 14061.091} C_VEL
LIN {X 0,Y 287.331,Z 559.714,A -85,B 0,C 180,E1 14060.61,E2 14060.61} C_VEL
LIN {X 0,Y 280.551,Z 576.326,A -85,B 0,C 180,E1 14059.335,E2 14059.335} C_VEL
LIN {X 0,Y 278.807,Z 583.098,A -85,B 0,C 180,E1 14058.635,E2 14058.635} C_VEL
LIN {X 0,Y 278.705,Z 584.045,A -85,B 0,C 180,E1 14058.522,E2 14058.522} C_VEL
LIN {X 0,Y 277.445,Z 599.064,A -85,B 0,C 180,E1 14056.537,E2 14056.537} C_VEL
LIN {X 0,Y 276.261,Z 612.924,A -85,B 0,C 180,E1 14054.244,E2 14054.244} C_VEL
LIN {X 0,Y 275.292,Z 625.067,A -85,B 0,C 180,E1 14051.732,E2 14051.732} C_VEL
LIN {X 0,Y 274.646,Z 634.813,A -85,B 0,C 180,E1 14049.214,E2 14049.214} C_VEL
LIN {X 0,Y 274.257,Z 643.879,A -85,B 0,C 180,E1 14046.276,E2 14046.276} C_VEL
LIN {X 0,Y 274.232,Z 651.211,A -85,B 0,C 180,E1 14043.132,E2 14043.132} C_VEL
LIN {X 0,Y 274.568,Z 656.118,A -85,B 0,C 180,E1 14040.206,E2 14040.206} C_VEL
LIN {X 0,Y 275.342,Z 659.521,A -85,B 0,C 180,E1 14037.083,E2 14037.083} C_VEL
LIN {X 0,Y 276.508,Z 661.032,A -85,B 0,C 180,E1 14034.186,E2 14034.186} C_VEL
LIN {X 0,Y 278.281,Z 660.871,A -85,B 0,C 180,E1 14031.11,E2 14031.11} C_VEL
LIN {X 0,Y 280.664,Z 658.963,A -85,B 0,C 180,E1 14028.073,E2 14028.073} C_VEL
LIN {X 0,Y 283.674,Z 655.185,A -85,B 0,C 180,E1 14025.087,E2 14025.087} C_VEL
LIN {X 0,Y 287.351,Z 649.554,A -85,B 0,C 180,E1 14022.167,E2 14022.167} C_VEL
LIN {X 0,Y 291.686,Z 641.84,A -85,B 0,C 180,E1 14019.322,E2 14019.322} C_VEL
LIN {X 0,Y 296.351,Z 632.619,A -85,B 0,C 180,E1 14016.747,E2 14016.747} C_VEL
LIN {X 0,Y 301.618,Z 621.153,A -85,B 0,C 180,E1 14014.259,E2 14014.259} C_VEL
LIN {X 0,Y 307.313,Z 607.403,A -85,B 0,C 180,E1 14011.954,E2 14011.954} C_VEL
LIN {X 0,Y 312.878,Z 592.336,A -85,B 0,C 180,E1 14009.99,E2 14009.99} C_VEL
LIN {X 0,Y 317.921,Z 576.934,A -85,B 0,C 180,E1 14008.421,E2 14008.421} C_VEL
LIN {X 0,Y 322.511,Z 560.631,A -85,B 0,C 180,E1 14007.141,E2 14007.141} C_VEL
LIN {X 0,Y 327.264,Z 539.889,A -85,B 0,C 180,E1 14005.951,E2 14005.951} C_VEL
LIN {X 0,Y 344.757,Z 466.179,A -85,B 0,C 180,E1 14002.583,E2 14002.583} C_VEL
LIN {X 0,Y 347.494,Z 452.376,A -85,B 0,C 180,E1 14000.805,E2 14000.805} C_VEL
LIN {X 0,Y 350.189,Z 441.695,A -85,B 0,C 180,E1 13999.139,E2 13999.139} C_VEL
LIN {X 0,Y 350.885,Z 440.842,A -85,B 0,C 180,E1 13997.739,E2 13997.739} C_VEL
LIN {X 0,Y 350.971,Z 440.995,A -85,B 0,C 180,E1 13997.535,E2 13997.535} C_VEL
LIN {X 0,Y 334.728,Z 512.988,A -85,B 0,C 180,E1 13994.887,E2 13994.887} C_VEL
LIN {X 0,Y 322.895,Z 573.936,A -85,B 0,C 180,E1 13992.534,E2 13992.534} C_VEL
LIN {X 0,Y 317.742,Z 593.847,A -85,B 0,C 180,E1 13991.484,E2 13991.484} C_VEL
LIN {X 0,Y 312.165,Z 612.054,A -85,B 0,C 180,E1 13990.197,E2 13990.197} C_VEL
LIN {X 0,Y 306.182,Z 629.286,A -85,B 0,C 180,E1 13988.59,E2 13988.59} C_VEL
LIN {X 0,Y 299.798,Z 646.39,A -85,B 0,C 180,E1 13986.525,E2 13986.525} C_VEL
LIN {X 0,Y 293.565,Z 662.381,A -85,B 0,C 180,E1 13984.076,E2 13984.076} C_VEL
LIN {X 0,Y 287.766,Z 676.898,A -85,B 0,C 180,E1 13981.266,E2 13981.266} C_VEL
LIN {X 0,Y 282.605,Z 690.157,A -85,B 0,C 180,E1 13978.072,E2 13978.072} C_VEL
LIN {X 0,Y 278.473,Z 701.689,A -85,B 0,C 180,E1 13974.615,E2 13974.615} C_VEL
LIN {X 0,Y 275.37,Z 711.742,A -85,B 0,C 180,E1 13970.846,E2 13970.846} C_VEL
LIN {X 0,Y 273.443,Z 720.144,A -85,B 0,C 180,E1 13966.792,E2 13966.792} C_VEL
LIN {X 0,Y 272.751,Z 726.528,A -85,B 0,C 180,E1 13962.708,E2 13962.708} C_VEL
LIN {X 0,Y 273.011,Z 730.75,A -85,B 0,C 180,E1 13958.85,E2 13958.85} C_VEL
LIN {X 0,Y 273.731,Z 733.079,A -85,B 0,C 180,E1 13955.241,E2 13955.241} C_VEL
LIN {X 0,Y 274.398,Z 733.731,A -85,B 0,C 180,E1 13952.09,E2 13952.09} C_VEL
LIN {X 0,Y 274.677,Z 733.026,A -85,B 0,C 180,E1 13949.167,E2 13949.167} C_VEL
LIN {X 0,Y 274.485,Z 730.935,A -85,B 0,C 180,E1 13946.242,E2 13946.242} C_VEL
LIN {X 0,Y 273.995,Z 727.098,A -85,B 0,C 180,E1 13943.028,E2 13943.028} C_VEL
LIN {X 0,Y 273.585,Z 721.354,A -85,B 0,C 180,E1 13939.686,E2 13939.686} C_VEL
LIN {X 0,Y 273.561,Z 713.526,A -85,B 0,C 180,E1 13936.258,E2 13936.258} C_VEL
LIN {X 0,Y 274.046,Z 704.146,A -85,B 0,C 180,E1 13933.031,E2 13933.031} C_VEL
LIN {X 0,Y 275.07,Z 693.333,A -85,B 0,C 180,E1 13930.022,E2 13930.022} C_VEL
LIN {X 0,Y 276.573,Z 680.903,A -85,B 0,C 180,E1 13927.205,E2 13927.205} C_VEL
LIN {X 0,Y 278.503,Z 666.805,A -85,B 0,C 180,E1 13924.597,E2 13924.597} C_VEL
LIN {X 0,Y 280.782,Z 650.794,A -85,B 0,C 180,E1 13922.195,E2 13922.195} C_VEL
LIN {X 0,Y 283.018,Z 634.56,A -85,B 0,C 180,E1 13920.242,E2 13920.242} C_VEL
LIN {X 0,Y 285.168,Z 617.474,A -85,B 0,C 180,E1 13918.625,E2 13918.625} C_VEL
LIN {X 0,Y 287.148,Z 599.58,A -85,B 0,C 180,E1 13917.338,E2 13917.338} C_VEL
LIN {X 0,Y 288.728,Z 580.317,A -85,B 0,C 180,E1 13916.345,E2 13916.345} C_VEL
LIN {X 0,Y 290.846,Z 534.317,A -85,B 0,C 180,E1 13914.845,E2 13914.845} C_VEL
LIN {X 0,Y 296.381,Z 422.743,A -85,B 0,C 180,E1 13911.326,E2 13911.326} C_VEL
LIN {X 0,Y 294.455,Z 390.669,A -85,B 0,C 180,E1 13910.019,E2 13910.019} C_VEL
LIN {X 0,Y 296.189,Z 381.846,A -85,B 0,C 180,E1 13908.769,E2 13908.769} C_VEL
LIN {X 0,Y 289.553,Z 360.846,A -85,B 0,C 180,E1 13904.508,E2 13904.508} C_VEL
LIN {X 0,Y 282.958,Z 341.005,A -85,B 0,C 180,E1 13900.027,E2 13900.027} C_VEL
LIN {X 0,Y 276.594,Z 322.807,A -85,B 0,C 180,E1 13895.467,E2 13895.467} C_VEL
LIN {X 0,Y 274.439,Z 316.611,A -85,B 0,C 180,E1 13893.742,E2 13893.742} C_VEL
LIN {X 0,Y 274.421,Z 316.613,A -85,B 0,C 180,E1 13888.988,E2 13888.988} C_VEL
LIN {X 0,Y 274.431,Z 316.614,A -85,B 0,C 180,E1 13884.086,E2 13884.086} C_VEL
LIN {X 0,Y 274.439,Z 316.615,A -85,B 0,C 180,E1 13879.365,E2 13879.365} C_VEL
LIN {X 0,Y 274.42,Z 316.613,A -85,B 0,C 180,E1 13874.563,E2 13874.563} C_VEL
LIN {X 0,Y 274.44,Z 316.613,A -85,B 0,C 180,E1 13869.862,E2 13869.862} C_VEL
LIN {X 0,Y 274.435,Z 316.612,A -85,B 0,C 180,E1 13865.229,E2 13865.229} C_VEL
LIN {X 0,Y 274.422,Z 316.613,A -85,B 0,C 180,E1 13860.42,E2 13860.42} C_VEL
LIN {X 0,Y 274.445,Z 316.609,A -85,B 0,C 180,E1 13855.615,E2 13855.615} C_VEL
LIN {X 0,Y 274.432,Z 316.606,A -85,B 0,C 180,E1 13850.99,E2 13850.99} C_VEL
LIN {X 0,Y 274.433,Z 316.612,A -85,B 0,C 180,E1 13846.09,E2 13846.09} C_VEL
LIN {X 0,Y 274.449,Z 316.6,A -85,B 0,C 180,E1 13841.305,E2 13841.305} C_VEL
LIN {X 0,Y 274.43,Z 316.611,A -85,B 0,C 180,E1 13836.605,E2 13836.605} C_VEL
LIN {X 0,Y 274.452,Z 316.601,A -85,B 0,C 180,E1 13831.736,E2 13831.736} C_VEL
LIN {X 0,Y 274.45,Z 316.609,A -85,B 0,C 180,E1 13827.128,E2 13827.128} C_VEL
LIN {X 0,Y 274.434,Z 316.608,A -85,B 0,C 180,E1 13822.239,E2 13822.239} C_VEL
LIN {X 0,Y 274.453,Z 316.598,A -85,B 0,C 180,E1 13817.631,E2 13817.631} C_VEL
LIN {X 0,Y 274.447,Z 316.609,A -85,B 0,C 180,E1 13812.928,E2 13812.928} C_VEL
LIN {X 0,Y 274.44,Z 316.602,A -85,B 0,C 180,E1 13808.001,E2 13808.001} C_VEL
LIN {X 0,Y 274.464,Z 316.606,A -85,B 0,C 180,E1 13803.371,E2 13803.371} C_VEL
LIN {X 0,Y 274.444,Z 316.607,A -85,B 0,C 180,E1 13798.605,E2 13798.605} C_VEL
LIN {X 0,Y 274.447,Z 316.596,A -85,B 0,C 180,E1 13793.851,E2 13793.851} C_VEL
LIN {X 0,Y 274.464,Z 316.609,A -85,B 0,C 180,E1 13789.137,E2 13789.137} C_VEL
LIN {X 0,Y 274.439,Z 316.601,A -85,B 0,C 180,E1 13784.294,E2 13784.294} C_VEL
LIN {X 0,Y 274.462,Z 316.611,A -85,B 0,C 180,E1 13779.434,E2 13779.434} C_VEL
LIN {X 0,Y 274.452,Z 316.601,A -85,B 0,C 180,E1 13774.805,E2 13774.805} C_VEL
LIN {X 0,Y 274.446,Z 316.61,A -85,B 0,C 180,E1 13769.998,E2 13769.998} C_VEL
LIN {X 0,Y 274.467,Z 316.604,A -85,B 0,C 180,E1 13765.192,E2 13765.192} C_VEL
LIN {X 0,Y 274.452,Z 316.606,A -85,B 0,C 180,E1 13760.563,E2 13760.563} C_VEL
LIN {X 0,Y 274.456,Z 316.611,A -85,B 0,C 180,E1 13755.655,E2 13755.655} C_VEL
LIN {X 0,Y 274.468,Z 316.607,A -85,B 0,C 180,E1 13750.859,E2 13750.859} C_VEL
LIN {X 0,Y 274.451,Z 316.61,A -85,B 0,C 180,E1 13746.114,E2 13746.114} C_VEL
LIN {X 0,Y 274.48,Z 316.607,A -85,B 0,C 180,E1 13741.258,E2 13741.258} C_VEL
LIN {X 0,Y 274.46,Z 316.608,A -85,B 0,C 180,E1 13736.53,E2 13736.53} C_VEL
LIN {X 0,Y 274.458,Z 316.612,A -85,B 0,C 180,E1 13731.732,E2 13731.732} C_VEL
LIN {X 0,Y 274.459,Z 316.638,A -85,B 0,C 180,E1 13728.187,E2 13728.187} C_VEL
LIN {X 0,Y 279.21,Z 332.401,A -85,B 0,C 180,E1 13723.665,E2 13723.665} C_VEL
LIN {X 0,Y 283.71,Z 348.607,A -85,B 0,C 180,E1 13719.368,E2 13719.368} C_VEL
LIN {X 0,Y 287.84,Z 365.202,A -85,B 0,C 180,E1 13715.281,E2 13715.281} C_VEL
LIN {X 0,Y 288.575,Z 369.053,A -85,B 0,C 180,E1 13714.382,E2 13714.382} C_VEL
LIN {X 0,Y 284.058,Z 396.281,A -85,B 0,C 180,E1 13709.057,E2 13709.057} C_VEL
LIN {X 0,Y 283.436,Z 401.088,A -85,B 0,C 180,E1 13708.178,E2 13708.178} C_VEL
LIN {X 0,Y 287.091,Z 442.163,A -85,B 0,C 180,E1 13706.15,E2 13706.15} C_VEL
LIN {X 0,Y 281.951,Z 536.558,A -85,B 0,C 180,E1 13702.392,E2 13702.392} C_VEL
LIN {X 0,Y 280.959,Z 553.963,A -85,B 0,C 180,E1 13701.335,E2 13701.335} C_VEL
LIN {X 0,Y 279.798,Z 570.628,A -85,B 0,C 180,E1 13699.951,E2 13699.951} C_VEL
LIN {X 0,Y 278.705,Z 584.045,A -85,B 0,C 180,E1 13698.522,E2 13698.522} C_VEL
LIN {X 0,Y 277.176,Z 590.695,A -85,B 0,C 180,E1 13697.738,E2 13697.738} C_VEL
LIN {X 0,Y 270.59,Z 604.804,A -85,B 0,C 180,E1 13695.875,E2 13695.875} C_VEL
LIN {X 0,Y 268.624,Z 610.73,A -85,B 0,C 180,E1 13694.897,E2 13694.897} C_VEL
LIN {X 0,Y 268.391,Z 612.384,A -85,B 0,C 180,E1 13694.594,E2 13694.594} C_VEL
LIN {X 0,Y 267.394,Z 624.477,A -85,B 0,C 180,E1 13692.084,E2 13692.084} C_VEL
LIN {X 0,Y 266.706,Z 634.648,A -85,B 0,C 180,E1 13689.491,E2 13689.491} C_VEL
LIN {X 0,Y 266.286,Z 644.034,A -85,B 0,C 180,E1 13686.465,E2 13686.465} C_VEL
LIN {X 0,Y 266.232,Z 650.807,A -85,B 0,C 180,E1 13683.657,E2 13683.657} C_VEL
LIN {X 0,Y 266.568,Z 656.572,A -85,B 0,C 180,E1 13680.427,E2 13680.427} C_VEL
LIN {X 0,Y 267.286,Z 660.211,A -85,B 0,C 180,E1 13677.424,E2 13677.424} C_VEL
LIN {X 0,Y 268.664,Z 662.383,A -85,B 0,C 180,E1 13674.016,E2 13674.016} C_VEL
LIN {X 0,Y 270.558,Z 662.563,A -85,B 0,C 180,E1 13670.854,E2 13670.854} C_VEL
LIN {X 0,Y 273.285,Z 660.813,A -85,B 0,C 180,E1 13667.531,E2 13667.531} C_VEL
LIN {X 0,Y 276.539,Z 657.32,A -85,B 0,C 180,E1 13664.478,E2 13664.478} C_VEL
LIN {X 0,Y 280.775,Z 651.578,A -85,B 0,C 180,E1 13661.304,E2 13661.304} C_VEL
LIN {X 0,Y 285.462,Z 644.133,A -85,B 0,C 180,E1 13658.419,E2 13658.419} C_VEL
LIN {X 0,Y 290.78,Z 634.714,A -85,B 0,C 180,E1 13655.676,E2 13655.676} C_VEL
LIN {X 0,Y 296.543,Z 623.349,A -85,B 0,C 180,E1 13653.138,E2 13653.138} C_VEL
LIN {X 0,Y 302.418,Z 610.565,A -85,B 0,C 180,E1 13650.919,E2 13650.919} C_VEL
LIN {X 0,Y 308.359,Z 596.236,A -85,B 0,C 180,E1 13648.963,E2 13648.963} C_VEL
LIN {X 0,Y 313.974,Z 580.899,A -85,B 0,C 180,E1 13647.329,E2 13647.329} C_VEL
LIN {X 0,Y 319.1,Z 564.521,A -85,B 0,C 180,E1 13645.99,E2 13645.99} C_VEL
LIN {X 0,Y 323.692,Z 546.681,A -85,B 0,C 180,E1 13644.903,E2 13644.903} C_VEL
LIN {X 0,Y 343.093,Z 469.061,A -85,B 0,C 180,E1 13641.343,E2 13641.343} C_VEL
LIN {X 0,Y 346.17,Z 456.372,A -85,B 0,C 180,E1 13639.656,E2 13639.656} C_VEL
LIN {X 0,Y 348.187,Z 449.56,A -85,B 0,C 180,E1 13638.563,E2 13638.563} C_VEL
LIN {X 0,Y 331.383,Z 519.46,A -85,B 0,C 180,E1 13635.993,E2 13635.993} C_VEL
LIN {X 0,Y 320.059,Z 572.859,A -85,B 0,C 180,E1 13633.911,E2 13633.911} C_VEL
LIN {X 0,Y 314.5,Z 592.654,A -85,B 0,C 180,E1 13632.872,E2 13632.872} C_VEL
LIN {X 0,Y 308.285,Z 611.347,A -85,B 0,C 180,E1 13631.55,E2 13631.55} C_VEL
LIN {X 0,Y 301.653,Z 628.868,A -85,B 0,C 180,E1 13629.896,E2 13629.896} C_VEL
LIN {X 0,Y 294.633,Z 646.152,A -85,B 0,C 180,E1 13627.775,E2 13627.775} C_VEL
LIN {X 0,Y 288.176,Z 661.203,A -85,B 0,C 180,E1 13625.412,E2 13625.412} C_VEL
LIN {X 0,Y 281.954,Z 675.4,A -85,B 0,C 180,E1 13622.618,E2 13622.618} C_VEL
LIN {X 0,Y 276.1,Z 688.982,A -85,B 0,C 180,E1 13619.269,E2 13619.269} C_VEL
LIN {X 0,Y 271.532,Z 700.359,A -85,B 0,C 180,E1 13615.756,E2 13615.756} C_VEL
LIN {X 0,Y 268.025,Z 710.265,A -85,B 0,C 180,E1 13611.905,E2 13611.905} C_VEL
LIN {X 0,Y 265.747,Z 718.612,A -85,B 0,C 180,E1 13607.745,E2 13607.745} C_VEL
LIN {X 0,Y 264.816,Z 724.981,A -85,B 0,C 180,E1 13603.54,E2 13603.54} C_VEL
LIN {X 0,Y 264.979,Z 729.41,A -85,B 0,C 180,E1 13599.339,E2 13599.339} C_VEL
LIN {X 0,Y 265.728,Z 731.686,A -85,B 0,C 180,E1 13595.616,E2 13595.616} C_VEL
LIN {X 0,Y 266.515,Z 732.279,A -85,B 0,C 180,E1 13592.152,E2 13592.152} C_VEL
LIN {X 0,Y 266.826,Z 731.465,A -85,B 0,C 180,E1 13589.143,E2 13589.143} C_VEL
LIN {X 0,Y 266.596,Z 729.187,A -85,B 0,C 180,E1 13586.074,E2 13586.074} C_VEL
LIN {X 0,Y 266.086,Z 725.127,A -85,B 0,C 180,E1 13582.771,E2 13582.771} C_VEL
LIN {X 0,Y 265.677,Z 719.225,A -85,B 0,C 180,E1 13579.375,E2 13579.375} C_VEL
LIN {X 0,Y 265.668,Z 711.686,A -85,B 0,C 180,E1 13576.064,E2 13576.064} C_VEL
LIN {X 0,Y 266.185,Z 702.134,A -85,B 0,C 180,E1 13572.74,E2 13572.74} C_VEL
LIN {X 0,Y 267.273,Z 691.063,A -85,B 0,C 180,E1 13569.642,E2 13569.642} C_VEL
LIN {X 0,Y 268.875,Z 678.217,A -85,B 0,C 180,E1 13566.714,E2 13566.714} C_VEL
LIN {X 0,Y 270.973,Z 663.34,A -85,B 0,C 180,E1 13563.956,E2 13563.956} C_VEL
LIN {X 0,Y 273.258,Z 647.585,A -85,B 0,C 180,E1 13561.599,E2 13561.599} C_VEL
LIN {X 0,Y 275.605,Z 630.701,A -85,B 0,C 180,E1 13559.598,E2 13559.598} C_VEL
LIN {X 0,Y 277.853,Z 612.848,A -85,B 0,C 180,E1 13557.944,E2 13557.944} C_VEL
LIN {X 0,Y 279.813,Z 594.744,A -85,B 0,C 180,E1 13556.683,E2 13556.683} C_VEL
LIN {X 0,Y 281.235,Z 575.99,A -85,B 0,C 180,E1 13555.765,E2 13555.765} C_VEL
LIN {X 0,Y 288.942,Z 423.393,A -85,B 0,C 180,E1 13550.753,E2 13550.753} C_VEL
LIN {X 0,Y 287.1,Z 391.391,A -85,B 0,C 180,E1 13549.416,E2 13549.416} C_VEL
LIN {X 0,Y 287.267,Z 389.774,A -85,B 0,C 180,E1 13549.264,E2 13549.264} C_VEL
LIN {X 0,Y 288.433,Z 383.533,A -85,B 0,C 180,E1 13548.322,E2 13548.322} C_VEL
LIN {X 0,Y 282.104,Z 363.463,A -85,B 0,C 180,E1 13544.146,E2 13544.146} C_VEL
LIN {X 0,Y 275.708,Z 344.056,A -85,B 0,C 180,E1 13539.665,E2 13539.665} C_VEL
LIN {X 0,Y 269.522,Z 326.314,A -85,B 0,C 180,E1 13535.103,E2 13535.103} C_VEL
LIN {X 0,Y 266.478,Z 317.605,A -85,B 0,C 180,E1 13532.666,E2 13532.666} C_VEL
LIN {X 0,Y 266.498,Z 317.603,A -85,B 0,C 180,E1 13527.971,E2 13527.971} C_VEL
LIN {X 0,Y 266.49,Z 317.605,A -85,B 0,C 180,E1 13523.191,E2 13523.191} C_VEL
LIN {X 0,Y 266.491,Z 317.604,A -85,B 0,C 180,E1 13518.147,E2 13518.147} C_VEL
LIN {X 0,Y 266.504,Z 317.597,A -85,B 0,C 180,E1 13513.454,E2 13513.454} C_VEL
LIN {X 0,Y 266.479,Z 317.596,A -85,B 0,C 180,E1 13508.635,E2 13508.635} C_VEL
LIN {X 0,Y 266.497,Z 317.599,A -85,B 0,C 180,E1 13503.875,E2 13503.875} C_VEL
LIN {X 0,Y 266.498,Z 317.599,A -85,B 0,C 180,E1 13499.143,E2 13499.143} C_VEL
LIN {X 0,Y 266.489,Z 317.601,A -85,B 0,C 180,E1 13494.189,E2 13494.189} C_VEL
LIN {X 0,Y 266.506,Z 317.593,A -85,B 0,C 180,E1 13489.395,E2 13489.395} C_VEL
LIN {X 0,Y 266.488,Z 317.601,A -85,B 0,C 180,E1 13484.554,E2 13484.554} C_VEL
LIN {X 0,Y 266.511,Z 317.59,A -85,B 0,C 180,E1 13479.699,E2 13479.699} C_VEL
LIN {X 0,Y 266.509,Z 317.599,A -85,B 0,C 180,E1 13475.157,E2 13475.157} C_VEL
LIN {X 0,Y 266.492,Z 317.584,A -85,B 0,C 180,E1 13470.318,E2 13470.318} C_VEL
LIN {X 0,Y 266.514,Z 317.601,A -85,B 0,C 180,E1 13465.498,E2 13465.498} C_VEL
LIN {X 0,Y 266.495,Z 317.589,A -85,B 0,C 180,E1 13460.611,E2 13460.611} C_VEL
LIN {X 0,Y 266.509,Z 317.594,A -85,B 0,C 180,E1 13455.754,E2 13455.754} C_VEL
LIN {X 0,Y 266.515,Z 317.595,A -85,B 0,C 180,E1 13451.033,E2 13451.033} C_VEL
LIN {X 0,Y 266.498,Z 317.583,A -85,B 0,C 180,E1 13446.087,E2 13446.087} C_VEL
LIN {X 0,Y 266.529,Z 317.599,A -85,B 0,C 180,E1 13441.427,E2 13441.427} C_VEL
LIN {X 0,Y 266.509,Z 317.59,A -85,B 0,C 180,E1 13436.755,E2 13436.755} C_VEL
LIN {X 0,Y 266.508,Z 317.593,A -85,B 0,C 180,E1 13431.801,E2 13431.801} C_VEL
LIN {X 0,Y 266.519,Z 317.595,A -85,B 0,C 180,E1 13427.013,E2 13427.013} C_VEL
LIN {X 0,Y 266.502,Z 317.591,A -85,B 0,C 180,E1 13422.126,E2 13422.126} C_VEL
LIN {X 0,Y 266.536,Z 317.596,A -85,B 0,C 180,E1 13417.326,E2 13417.326} C_VEL
LIN {X 0,Y 266.505,Z 317.594,A -85,B 0,C 180,E1 13412.364,E2 13412.364} C_VEL
LIN {X 0,Y 266.515,Z 317.598,A -85,B 0,C 180,E1 13407.633,E2 13407.633} C_VEL
LIN {X 0,Y 266.527,Z 317.597,A -85,B 0,C 180,E1 13402.887,E2 13402.887} C_VEL
LIN {X 0,Y 266.511,Z 317.596,A -85,B 0,C 180,E1 13397.871,E2 13397.871} C_VEL
LIN {X 0,Y 266.53,Z 317.594,A -85,B 0,C 180,E1 13393.209,E2 13393.209} C_VEL
LIN {X 0,Y 266.514,Z 317.596,A -85,B 0,C 180,E1 13388.427,E2 13388.427} C_VEL
LIN {X 0,Y 266.526,Z 317.6,A -85,B 0,C 180,E1 13383.484,E2 13383.484} C_VEL
LIN {X 0,Y 266.533,Z 317.595,A -85,B 0,C 180,E1 13378.786,E2 13378.786} C_VEL
LIN {X 0,Y 266.517,Z 317.601,A -85,B 0,C 180,E1 13373.757,E2 13373.757} C_VEL
LIN {X 0,Y 266.548,Z 317.651,A -85,B 0,C 180,E1 13369.16,E2 13369.16} C_VEL
LIN {X 0,Y 271.411,Z 333.777,A -85,B 0,C 180,E1 13364.381,E2 13364.381} C_VEL
LIN {X 0,Y 275.644,Z 349.008,A -85,B 0,C 180,E1 13360.211,E2 13360.211} C_VEL
LIN {X 0,Y 279.86,Z 365.73,A -85,B 0,C 180,E1 13355.961,E2 13355.961} C_VEL
LIN {X 0,Y 280.851,Z 371.132,A -85,B 0,C 180,E1 13354.674,E2 13354.674} C_VEL
LIN {X 0,Y 276.192,Z 398.226,A -85,B 0,C 180,E1 13349.252,E2 13349.252} C_VEL
LIN {X 0,Y 275.863,Z 400.986,A -85,B 0,C 180,E1 13348.767,E2 13348.767} C_VEL
LIN {X 0,Y 279.467,Z 442.809,A -85,B 0,C 180,E1 13346.64,E2 13346.64} C_VEL
LIN {X 0,Y 274.114,Z 537.36,A -85,B 0,C 180,E1 13342.721,E2 13342.721} C_VEL
LIN {X 0,Y 273.096,Z 554.665,A -85,B 0,C 180,E1 13341.636,E2 13341.636} C_VEL
LIN {X 0,Y 271.838,Z 572.141,A -85,B 0,C 180,E1 13340.132,E2 13340.132} C_VEL
LIN {X 0,Y 270.482,Z 588.368,A -85,B 0,C 180,E1 13338.309,E2 13338.309} C_VEL
LIN {X 0,Y 269.131,Z 603.984,A -85,B 0,C 180,E1 13336.064,E2 13336.064} C_VEL
LIN {X 0,Y 268.391,Z 612.384,A -85,B 0,C 180,E1 13334.594,E2 13334.594} C_VEL
LIN {X 0,Y 266.939,Z 618.15,A -85,B 0,C 180,E1 13333.522,E2 13333.522} C_VEL
LIN {X 0,Y 261.761,Z 627.945,A -85,B 0,C 180,E1 13331.473,E2 13331.473} C_VEL
LIN {X 0,Y 259.184,Z 633.519,A -85,B 0,C 180,E1 13330.043,E2 13330.043} C_VEL
LIN {X 0,Y 258.664,Z 636.184,A -85,B 0,C 180,E1 13329.262,E2 13329.262} C_VEL
LIN {X 0,Y 258.27,Z 645.892,A -85,B 0,C 180,E1 13325.997,E2 13325.997} C_VEL
LIN {X 0,Y 258.295,Z 652.975,A -85,B 0,C 180,E1 13322.876,E2 13322.876} C_VEL
LIN {X 0,Y 258.722,Z 658.258,A -85,B 0,C 180,E1 13319.775,E2 13319.775} C_VEL
LIN {X 0,Y 259.651,Z 661.975,A -85,B 0,C 180,E1 13316.465,E2 13316.465} C_VEL
LIN {X 0,Y 261.171,Z 663.954,A -85,B 0,C 180,E1 13313.181,E2 13313.181} C_VEL
LIN {X 0,Y 263.318,Z 664.104,A -85,B 0,C 180,E1 13309.938,E2 13309.938} C_VEL
LIN {X 0,Y 266.368,Z 662.367,A -85,B 0,C 180,E1 13306.539,E2 13306.539} C_VEL
LIN {X 0,Y 269.966,Z 658.919,A -85,B 0,C 180,E1 13303.428,E2 13303.428} C_VEL
LIN {X 0,Y 274.616,Z 653.291,A -85,B 0,C 180,E1 13300.205,E2 13300.205} C_VEL
LIN {X 0,Y 279.715,Z 645.992,A -85,B 0,C 180,E1 13297.288,E2 13297.288} C_VEL
LIN {X 0,Y 285.564,Z 636.661,A -85,B 0,C 180,E1 13294.488,E2 13294.488} C_VEL
LIN {X 0,Y 292.143,Z 624.933,A -85,B 0,C 180,E1 13291.813,E2 13291.813} C_VEL
LIN {X 0,Y 298.734,Z 611.878,A -85,B 0,C 180,E1 13289.529,E2 13289.529} C_VEL
LIN {X 0,Y 305.119,Z 597.797,A -85,B 0,C 180,E1 13287.601,E2 13287.601} C_VEL
LIN {X 0,Y 311.428,Z 582.032,A -85,B 0,C 180,E1 13285.925,E2 13285.925} C_VEL
LIN {X 0,Y 317.203,Z 564.902,A -85,B 0,C 180,E1 13284.548,E2 13284.548} C_VEL
LIN {X 0,Y 322.115,Z 546.949,A -85,B 0,C 180,E1 13283.485,E2 13283.485} C_VEL
LIN {X 0,Y 341.846,Z 472.283,A -85,B 0,C 180,E1 13280.111,E2 13280.111} C_VEL
LIN {X 0,Y 343.459,Z 466.404,A -85,B 0,C 180,E1 13279.321,E2 13279.321} C_VEL
LIN {X 0,Y 326.764,Z 532.774,A -85,B 0,C 180,E1 13276.87,E2 13276.87} C_VEL
LIN {X 0,Y 317.734,Z 571.857,A -85,B 0,C 180,E1 13275.333,E2 13275.333} C_VEL
LIN {X 0,Y 311.538,Z 592.175,A -85,B 0,C 180,E1 13274.273,E2 13274.273} C_VEL
LIN {X 0,Y 304.982,Z 610.29,A -85,B 0,C 180,E1 13272.995,E2 13272.995} C_VEL
LIN {X 0,Y 297.96,Z 627.47,A -85,B 0,C 180,E1 13271.383,E2 13271.383} C_VEL
LIN {X 0,Y 290.447,Z 644.452,A -85,B 0,C 180,E1 13269.304,E2 13269.304} C_VEL
LIN {X 0,Y 283.248,Z 659.815,A -85,B 0,C 180,E1 13266.879,E2 13266.879} C_VEL
LIN {X 0,Y 276.096,Z 674.649,A -85,B 0,C 180,E1 13263.898,E2 13263.898} C_VEL
LIN {X 0,Y 269.758,Z 687.969,A -85,B 0,C 180,E1 13260.518,E2 13260.518} C_VEL
LIN {X 0,Y 264.714,Z 699.145,A -85,B 0,C 180,E1 13256.946,E2 13256.946} C_VEL
LIN {X 0,Y 260.787,Z 708.862,A -85,B 0,C 180,E1 13253.023,E2 13253.023} C_VEL
LIN {X 0,Y 258.127,Z 717.124,A -85,B 0,C 180,E1 13248.755,E2 13248.755} C_VEL
LIN {X 0,Y 256.921,Z 723.453,A -85,B 0,C 180,E1 13244.424,E2 13244.424} C_VEL
LIN {X 0,Y 256.92,Z 727.881,A -85,B 0,C 180,E1 13240.088,E2 13240.088} C_VEL
LIN {X 0,Y 257.657,Z 730.187,A -85,B 0,C 180,E1 13236.24,E2 13236.24} C_VEL
LIN {X 0,Y 258.542,Z 730.833,A -85,B 0,C 180,E1 13232.662,E2 13232.662} C_VEL
LIN {X 0,Y 258.977,Z 730.075,A -85,B 0,C 180,E1 13229.559,E2 13229.559} C_VEL
LIN {X 0,Y 258.808,Z 727.897,A -85,B 0,C 180,E1 13226.458,E2 13226.458} C_VEL
LIN {X 0,Y 258.275,Z 723.953,A -85,B 0,C 180,E1 13223.109,E2 13223.109} C_VEL
LIN {X 0,Y 257.828,Z 718.317,A -85,B 0,C 180,E1 13219.726,E2 13219.726} C_VEL
LIN {X 0,Y 257.762,Z 710.871,A -85,B 0,C 180,E1 13216.315,E2 13216.315} C_VEL
LIN {X 0,Y 258.231,Z 701.416,A -85,B 0,C 180,E1 13212.888,E2 13212.888} C_VEL
LIN {X 0,Y 259.291,Z 690.456,A -85,B 0,C 180,E1 13209.695,E2 13209.695} C_VEL
LIN {X 0,Y 260.916,Z 677.5,A -85,B 0,C 180,E1 13206.635,E2 13206.635} C_VEL
LIN {X 0,Y 263.053,Z 662.577,A -85,B 0,C 180,E1 13203.775,E2 13203.775} C_VEL
LIN {X 0,Y 265.312,Z 647.291,A -85,B 0,C 180,E1 13201.407,E2 13201.407} C_VEL
LIN {X 0,Y 267.693,Z 630.549,A -85,B 0,C 180,E1 13199.345,E2 13199.345} C_VEL
LIN {X 0,Y 270.064,Z 612.16,A -85,B 0,C 180,E1 13197.582,E2 13197.582} C_VEL
LIN {X 0,Y 272.094,Z 593.785,A -85,B 0,C 180,E1 13196.262,E2 13196.262} C_VEL
LIN {X 0,Y 273.529,Z 575.123,A -85,B 0,C 180,E1 13195.324,E2 13195.324} C_VEL
LIN {X 0,Y 281.493,Z 424.096,A -85,B 0,C 180,E1 13190.176,E2 13190.176} C_VEL
LIN {X 0,Y 279.745,Z 392.127,A -85,B 0,C 180,E1 13188.797,E2 13188.797} C_VEL
LIN {X 0,Y 279.811,Z 390.351,A -85,B 0,C 180,E1 13188.689,E2 13188.689} C_VEL
LIN {X 0,Y 280.839,Z 385.764,A -85,B 0,C 180,E1 13187.987,E2 13187.987} C_VEL
LIN {X 0,Y 274.643,Z 366.028,A -85,B 0,C 180,E1 13183.768,E2 13183.768} C_VEL
LIN {X 0,Y 268.769,Z 347.986,A -85,B 0,C 180,E1 13179.508,E2 13179.508} C_VEL
LIN {X 0,Y 262.59,Z 330.134,A -85,B 0,C 180,E1 13174.834,E2 13174.834} C_VEL
LIN {X 0,Y 258.561,Z 318.588,A -85,B 0,C 180,E1 13171.473,E2 13171.473} C_VEL
LIN {X 0,Y 258.539,Z 318.59,A -85,B 0,C 180,E1 13166.658,E2 13166.658} C_VEL
LIN {X 0,Y 258.568,Z 318.593,A -85,B 0,C 180,E1 13161.794,E2 13161.794} C_VEL
LIN {X 0,Y 258.543,Z 318.589,A -85,B 0,C 180,E1 13156.864,E2 13156.864} C_VEL
LIN {X 0,Y 258.555,Z 318.589,A -85,B 0,C 180,E1 13151.946,E2 13151.946} C_VEL
LIN {X 0,Y 258.554,Z 318.591,A -85,B 0,C 180,E1 13147.111,E2 13147.111} C_VEL
LIN {X 0,Y 258.557,Z 318.587,A -85,B 0,C 180,E1 13141.998,E2 13141.998} C_VEL
LIN {X 0,Y 258.562,Z 318.582,A -85,B 0,C 180,E1 13137.344,E2 13137.344} C_VEL
LIN {X 0,Y 258.548,Z 318.589,A -85,B 0,C 180,E1 13132.448,E2 13132.448} C_VEL
LIN {X 0,Y 258.573,Z 318.587,A -85,B 0,C 180,E1 13127.497,E2 13127.497} C_VEL
LIN {X 0,Y 258.551,Z 318.584,A -85,B 0,C 180,E1 13122.68,E2 13122.68} C_VEL
LIN {X 0,Y 258.574,Z 318.586,A -85,B 0,C 180,E1 13117.735,E2 13117.735} C_VEL
LIN {X 0,Y 258.558,Z 318.582,A -85,B 0,C 180,E1 13112.797,E2 13112.797} C_VEL
LIN {X 0,Y 258.57,Z 318.583,A -85,B 0,C 180,E1 13107.754,E2 13107.754} C_VEL
LIN {X 0,Y 258.561,Z 318.585,A -85,B 0,C 180,E1 13102.804,E2 13102.804} C_VEL
LIN {X 0,Y 258.572,Z 318.573,A -85,B 0,C 180,E1 13097.719,E2 13097.719} C_VEL
LIN {X 0,Y 258.567,Z 318.587,A -85,B 0,C 180,E1 13092.886,E2 13092.886} C_VEL
LIN {X 0,Y 258.564,Z 318.576,A -85,B 0,C 180,E1 13087.928,E2 13087.928} C_VEL
LIN {X 0,Y 258.575,Z 318.585,A -85,B 0,C 180,E1 13082.963,E2 13082.963} C_VEL
LIN {X 0,Y 258.569,Z 318.586,A -85,B 0,C 180,E1 13077.896,E2 13077.896} C_VEL
LIN {X 0,Y 258.579,Z 318.578,A -85,B 0,C 180,E1 13072.986,E2 13072.986} C_VEL
LIN {X 0,Y 258.569,Z 318.588,A -85,B 0,C 180,E1 13067.977,E2 13067.977} C_VEL
LIN {X 0,Y 258.588,Z 318.574,A -85,B 0,C 180,E1 13063.185,E2 13063.185} C_VEL
LIN {X 0,Y 258.564,Z 318.588,A -85,B 0,C 180,E1 13058.164,E2 13058.164} C_VEL
LIN {X 0,Y 258.582,Z 318.578,A -85,B 0,C 180,E1 13053.323,E2 13053.323} C_VEL
LIN {X 0,Y 258.569,Z 318.586,A -85,B 0,C 180,E1 13048.447,E2 13048.447} C_VEL
LIN {X 0,Y 258.594,Z 318.587,A -85,B 0,C 180,E1 13043.337,E2 13043.337} C_VEL
LIN {X 0,Y 258.57,Z 318.584,A -85,B 0,C 180,E1 13038.398,E2 13038.398} C_VEL
LIN {X 0,Y 258.584,Z 318.582,A -85,B 0,C 180,E1 13033.508,E2 13033.508} C_VEL
LIN {X 0,Y 258.584,Z 318.584,A -85,B 0,C 180,E1 13028.685,E2 13028.685} C_VEL
LIN {X 0,Y 258.584,Z 318.588,A -85,B 0,C 180,E1 13023.596,E2 13023.596} C_VEL
LIN {X 0,Y 258.594,Z 318.584,A -85,B 0,C 180,E1 13018.792,E2 13018.792} C_VEL
LIN {X 0,Y 258.58,Z 318.589,A -85,B 0,C 180,E1 13013.727,E2 13013.727} C_VEL
LIN {X 0,Y 258.576,Z 318.59,A -85,B 0,C 180,E1 13010.21,E2 13010.21} C_VEL
LIN {X 0,Y 263.153,Z 333.613,A -85,B 0,C 180,E1 13005.581,E2 13005.581} C_VEL
LIN {X 0,Y 267.588,Z 349.33,A -85,B 0,C 180,E1 13001.115,E2 13001.115} C_VEL
LIN {X 0,Y 271.656,Z 365.515,A -85,B 0,C 180,E1 12996.861,E2 12996.861} C_VEL
LIN {X 0,Y 273.205,Z 372.763,A -85,B 0,C 180,E1 12995.066,E2 12995.066} C_VEL
LIN {X 0,Y 268.415,Z 399.596,A -85,B 0,C 180,E1 12989.571,E2 12989.571} C_VEL
LIN {X 0,Y 268.316,Z 401.123,A -85,B 0,C 180,E1 12989.364,E2 12989.364} C_VEL
LIN {X 0,Y 271.814,Z 443.59,A -85,B 0,C 180,E1 12987.127,E2 12987.127} C_VEL
LIN {X 0,Y 266.285,Z 538.187,A -85,B 0,C 180,E1 12983.067,E2 12983.067} C_VEL
LIN {X 0,Y 265.204,Z 555.919,A -85,B 0,C 180,E1 12981.912,E2 12981.912} C_VEL
LIN {X 0,Y 263.933,Z 572.889,A -85,B 0,C 180,E1 12980.393,E2 12980.393} C_VEL
LIN {X 0,Y 262.483,Z 589.707,A -85,B 0,C 180,E1 12978.428,E2 12978.428} C_VEL
LIN {X 0,Y 261.105,Z 605.197,A -85,B 0,C 180,E1 12976.115,E2 12976.115} C_VEL
LIN {X 0,Y 259.874,Z 619.322,A -85,B 0,C 180,E1 12973.457,E2 12973.457} C_VEL
LIN {X 0,Y 258.919,Z 631.957,A -85,B 0,C 180,E1 12970.454,E2 12970.454} C_VEL
LIN {X 0,Y 258.664,Z 636.184,A -85,B 0,C 180,E1 12969.262,E2 12969.262} C_VEL
LIN {X 0,Y 257.443,Z 640.66,A -85,B 0,C 180,E1 12967.876,E2 12967.876} C_VEL
LIN {X 0,Y 252.45,Z 648.66,A -85,B 0,C 180,E1 12965.06,E2 12965.06} C_VEL
LIN {X 0,Y 250.491,Z 652.696,A -85,B 0,C 180,E1 12963.298,E2 12963.298} C_VEL
LIN {X 0,Y 250.336,Z 654.067,A -85,B 0,C 180,E1 12962.603,E2 12962.603} C_VEL
LIN {X 0,Y 250.849,Z 659.568,A -85,B 0,C 180,E1 12959.312,E2 12959.312} C_VEL
LIN {X 0,Y 251.907,Z 663.385,A -85,B 0,C 180,E1 12955.9,E2 12955.9} C_VEL
LIN {X 0,Y 253.603,Z 665.443,A -85,B 0,C 180,E1 12952.521,E2 12952.521} C_VEL
LIN {X 0,Y 255.979,Z 665.722,A -85,B 0,C 180,E1 12949.191,E2 12949.191} C_VEL
LIN {X 0,Y 259.322,Z 664.133,A -85,B 0,C 180,E1 12945.711,E2 12945.711} C_VEL
LIN {X 0,Y 263.245,Z 660.901,A -85,B 0,C 180,E1 12942.536,E2 12942.536} C_VEL
LIN {X 0,Y 268.262,Z 655.499,A -85,B 0,C 180,E1 12939.26,E2 12939.26} C_VEL
LIN {X 0,Y 273.758,Z 648.555,A -85,B 0,C 180,E1 12936.309,E2 12936.309} C_VEL
LIN {X 0,Y 280.455,Z 638.958,A -85,B 0,C 180,E1 12933.305,E2 12933.305} C_VEL
LIN {X 0,Y 287.502,Z 627.597,A -85,B 0,C 180,E1 12930.633,E2 12930.633} C_VEL
LIN {X 0,Y 294.536,Z 615.06,A -85,B 0,C 180,E1 12928.364,E2 12928.364} C_VEL
LIN {X 0,Y 301.624,Z 601.037,A -85,B 0,C 180,E1 12926.384,E2 12926.384} C_VEL
LIN {X 0,Y 308.604,Z 585.188,A -85,B 0,C 180,E1 12924.665,E2 12924.665} C_VEL
LIN {X 0,Y 314.708,Z 568.851,A -85,B 0,C 180,E1 12923.321,E2 12923.321} C_VEL
LIN {X 0,Y 319.976,Z 551.543,A -85,B 0,C 180,E1 12922.261,E2 12922.261} C_VEL
LIN {X 0,Y 335.536,Z 494.968,A -85,B 0,C 180,E1 12919.678,E2 12919.678} C_VEL
LIN {X 0,Y 316.097,Z 570.452,A -85,B 0,C 180,E1 12916.813,E2 12916.813} C_VEL
LIN {X 0,Y 309.223,Z 591.341,A -85,B 0,C 180,E1 12915.744,E2 12915.744} C_VEL
LIN {X 0,Y 302.32,Z 608.972,A -85,B 0,C 180,E1 12914.521,E2 12914.521} C_VEL
LIN {X 0,Y 294.554,Z 626.539,A -85,B 0,C 180,E1 12912.892,E2 12912.892} C_VEL
LIN {X 0,Y 286.859,Z 642.541,A -85,B 0,C 180,E1 12910.943,E2 12910.943} C_VEL
LIN {X 0,Y 279.097,Z 657.728,A -85,B 0,C 180,E1 12908.563,E2 12908.563} C_VEL
LIN {X 0,Y 271.318,Z 672.427,A -85,B 0,C 180,E1 12905.611,E2 12905.611} C_VEL
LIN {X 0,Y 264.312,Z 685.662,A -85,B 0,C 180,E1 12902.236,E2 12902.236} C_VEL
LIN {X 0,Y 258.637,Z 696.813,A -85,B 0,C 180,E1 12898.646,E2 12898.646} C_VEL
LIN {X 0,Y 254.027,Z 706.716,A -85,B 0,C 180,E1 12894.597,E2 12894.597} C_VEL
LIN {X 0,Y 250.84,Z 714.926,A -85,B 0,C 180,E1 12890.293,E2 12890.293} C_VEL
LIN {X 0,Y 249.116,Z 721.699,A -85,B 0,C 180,E1 12885.569,E2 12885.569} C_VEL
LIN {X 0,Y 248.863,Z 726.155,A -85,B 0,C 180,E1 12881.121,E2 12881.121} C_VEL
LIN {X 0,Y 249.577,Z 728.669,A -85,B 0,C 180,E1 12876.905,E2 12876.905} C_VEL
LIN {X 0,Y 250.549,Z 729.354,A -85,B 0,C 180,E1 12873.204,E2 12873.204} C_VEL
LIN {X 0,Y 251.127,Z 728.646,A -85,B 0,C 180,E1 12870.002,E2 12870.002} C_VEL
LIN {X 0,Y 251.035,Z 726.701,A -85,B 0,C 180,E1 12867.034,E2 12867.034} C_VEL
LIN {X 0,Y 250.502,Z 722.885,A -85,B 0,C 180,E1 12863.585,E2 12863.585} C_VEL
LIN {X 0,Y 249.998,Z 717.343,A -85,B 0,C 180,E1 12860.099,E2 12860.099} C_VEL
LIN {X 0,Y 249.872,Z 709.81,A -85,B 0,C 180,E1 12856.506,E2 12856.506} C_VEL
LIN {X 0,Y 250.29,Z 700.607,A -85,B 0,C 180,E1 12853.047,E2 12853.047} C_VEL
